# B&R Automation Studio project RobotComau
Automation Studio 4.11.3.51 SP; technology packages: mapp 5.18.0, mappCockpit 5.18.0, mappMotion 5.18.1, mappView 5.18.1, mappVision 5.18.0

## Configuration Config1

CPU 5APC3100.KBU1-000, AutomationRuntime B4.92, Build 4.1.2, Safety 0.0, Vc V4.72.5

### Task classes (Cpu.sw)
```
Cyclic#1 (cycle 2000 us, tolerance 0 us):
  OpcCtrl <- Services.OpcCtrl.prg
  ComauManua <- Robot.PackML.PackML_Manual.prg
  PackML_Aut <- Robot.PackML.PackML_Auto.prg
  PackML_Log <- Robot.PackML.PackML_Logic.prg
  PackML_Sem <- Robot.PackML.PackML_SemiAuto.prg
  RobotMove <- (binary)
Cyclic#2:
  File_explo <- Services.File_explorer.prg
Cyclic#4:
  Alarms <- Services.Alarms.prg
  Elements_d <- Camera.Elements_detection.prg
  Recipe <- Robot.Recipe.prg
  AuditProgr <- Services.AuditPckg.AuditProgram.prg
  AlarmClear <- Services.AlarmClearHistory.prg
DataObjects: McAcpSys
NcDataObjects: McDriveLog
Binaries: McAcpDrv, udbdef, McAcpSim, mvLoader, arflatprv, McPathXT, TCData, visionUnit, mCoWebSc, McMechSys, FWRules, arcoal, arsvcreg, TCLang, Settings, iomap, Config_3, Settings_1, viComp, Config_4, Role, ashwac, Hierarchy, asfw, Config_5, sysconf, Config_2, arconfig, Config_1, ashwd, User, Config_6, Config, Config_7, Config_9, PixelCount, Config_8, Config_13, Config_11, Config_14, Config_12, Config_10, TC, viApp, Matching15
Libraries: McBase, ViBase, AsZip, FileIO, AsARCfg, powerlnk, AsEPL, AsIO, sys_lib, astime, runtime, MpRobotics, McAxGroup, MpBase, McPathGen, McAxis, McProgInt, McAcpAx, CoTrace, standard, MpAlarmX, MpUserX, AsArSdm, MpRecipe, MpAudit, asarprof, asieccon, asarlog, asmem, brsystem, dataobj, arssl, asopcuac, aseth, ashw, arcert, aruser, asbrstr, mpfile, asusb, MpPackML, MpServer, MpWebXs
```

### Hardware
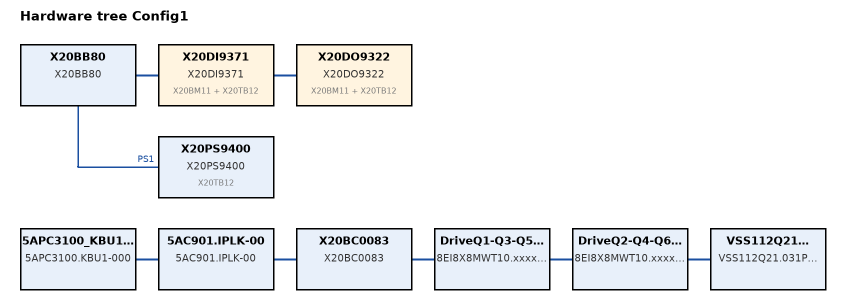
```
5AC901.IPLK-00 : 5AC901.IPLK-00 v1.8.0.1  [SL -> 5APC3100_KBU1_000.SL2]
  Connector IF1:
    MtuSize = 1500
    CycleTime = 400
    Channel1
    ChannelID1 = McAcpBroadcast
    ChannelType1 = OCTET[200]
    InternetAddress = 192.168.200.240
    SubnetMask = 255.255.255.0
5APC3100_KBU1_000 : 5APC3100.KBU1-000 v2.2.1.0
  Connector IF3:
    AssignedOperatingSystem = ARemb
    ActivateDevice = 1
    Mode = Manual
    InternetAddress = 192.168.0.10
    SubnetMask = 255.255.255.0
    InaPort = 81
    ActivateSnmp = 2
  Connector IF4:
    AssignedOperatingSystem = ARemb
    ActivateDevice = 1
  Connector IF5:
    AssignedOperatingSystem = ARemb
  Connector IF6:
    AssignedOperatingSystem = ARemb
  Connector IF7:
    AssignedOperatingSystem = ARemb
  Connector IF8:
    AssignedOperatingSystem = ARemb
  ConfigurationID = RobotComau_Config1
  RemMemDevice = PCI.2.IPLK.SRAM
  RemMemSize = 1024
  PermanentPvSize = 512
  RemanentGlobalPvSize = 512
  TimerDeviceType = EPLX2X
  TimerDevice = 5AC901.IPLK-00.IF1
  TaskClassIdleTime = 2000
  Cyclic1Duration = 2000
  Cyclic1Tolerance = 0
  FileDevice1
  FileDeviceName1 = CNC_PrgDir
  FileDevicePath1 = F:\RobotProgram
  FileDevice2
  FileDeviceName2 = RecipeDir
  FileDevicePath2 = F:\Data
  FileDevice3
  FileDeviceName3 = AuditDir
  FileDevicePath3 = F:\Audit
  FileDevice4
  FileDeviceName4 = FilesDir
  FileDevicePath4 = F:\
  FtpUser1
  FtpUsername1 = admin
  FtpUserPassword1 = QCzPEyxrRcQJkbJUmFYJydudCaTwVAMxyUFRcNQN44M=
  FtpUserSalt1 = 07CFXo9y
  FTPAccessRight1 = 0
  ActivateOpcUa = 1
  OpcUaActivateAuditEvents = 1
  OpcUa_Security_AdminRole = Administrators
  OpcUaInformationModels_PV_Version = 1
DriveQ1-Q3-Q5_Racer3_1 : 8EI8X8MWT10.xxxx-1 v2.3.1.1  [PLK1 -> X20BC0083.PLK2 (NodeNumber=4) [Cable Type=PowerlinkCable, Length=10, Version=1.0.0.3]; PLK2 -> DriveQ2-Q4-Q6_Racer3_1.PLK1 (NodeNumber=4) [Cable Type=PowerlinkCable, Length=10, Version=1.0.0.3]]
  DriveConfiguration/Module:
    McAcoposTypeID = AcoposP3TConfig
    ActivateACOPOSSimulationOnPLC = 0
  DriveConfiguration/Encoder/EncoderX41:
    InterfaceType = EnDat
  DriveConfiguration/Encoder/EncoderX42:
    InterfaceType = EnDat
  DriveConfiguration/Encoder/EncoderX43:
    InterfaceType = EnDat
  DriveConfiguration/Channel[1]/RealAxis:
    AxisReference = gAxisQ1_Racer3_1
    MechanicalElementsIsInvisible = 0
  DriveConfiguration/Channel[1]/RealAxis/MechanicalElements/Gearbox:
    InputIsReadOnly = 1
    Input = 81818
    OutputIsReadOnly = 1
    Output = 1000
  DriveConfiguration/Channel[1]/RealAxis/MechanicalElements/RotaryToLinearTransformation:
    ReferenceDistanceIsReadOnly = 1
    ReferenceDistance = 360
  DriveConfiguration/Channel[1]/RealAxis/Controller:
    ModeIsReadOnly = 1
    Mode = PositionControllerWithTorqueFeedForward
  DriveConfiguration/Channel[1]/RealAxis/Controller/Mode/Position:
    ProportionalGainIsReadOnly = 1
    ProportionalGain = 75.0
    IntegrationTimeIsReadOnly = 1
    IntegrationTime = 0.0
    TotalDelayTime = 0.0004
  DriveConfiguration/Channel[1]/RealAxis/Controller/Mode/Speed:
    ProportionalGainIsReadOnly = 1
    ProportionalGain = 2.0
    IntegrationTimeIsReadOnly = 1
    IntegrationTime = 0.0
    FilterTimeIsReadOnly = 1
    FilterTime = 0.0008
  DriveConfiguration/Channel[1]/RealAxis/Controller/Mode:
    FeedForwardIsReadOnly = 1
    FeedForward = CyclicValueFromAxesGroup
  DriveConfiguration/Channel[1]/RealAxis/Controller/Mode/LoopFilters:
    LoopFilterXIsReadOnly = 0
    LoopFilter1 = NotUsed
    LoopFilter2 = NotUsed
    LoopFilter3 = NotUsed
  DriveConfiguration/Channel[1]/RealAxis/Homing:
    ModeIsReadOnly = 0
    Mode = RestorePosition
    RestorePositionVariable = ::RestorePos[0]
  DriveConfiguration/Channel[1]/RealAxis/StopReaction:
    QuickstopIsReadOnly = 0
    Quickstop = DecelerationLimit
    DriveErrorIsReadOnly = 0
    DriveError = DecelerationLimit
  DriveConfiguration/Channel[1]/RealAxis/MovementErrorLimits:
    PositionError = 1.0
    VelocityErrorMonitoring = Automatic1
  DriveConfiguration/Channel[1]/RealAxis:
    JerkFilterIsReadOnly = 0
    JerkFilter = Used
  DriveConfiguration/Channel[1]/RealAxis/JerkFilter:
    JerkTimeMin = 0
    JerkTime = 0.01
  DriveConfiguration/Channel[1]/RealAxis/DigitalInputs/HomingSwitch:
    SourceIsReadOnly = 0
    Source = NotUsed
    Level = High
  DriveConfiguration/Channel[1]/RealAxis/DigitalInputs/PositiveLimitSwitch:
    SourceIsReadOnly = 0
    Source = NotUsed
    Level = High
  DriveConfiguration/Channel[1]/RealAxis/DigitalInputs/NegativeLimitSwitch:
    SourceIsReadOnly = 0
    Source = NotUsed
    Level = High
  DriveConfiguration/Channel[1]/RealAxis/DigitalInputs/Trigger1:
    Source = X8Trigger1
    Level = High
  DriveConfiguration/Channel[1]/RealAxis/DigitalInputs/Trigger2:
    Source = X8Trigger2
    Level = High
  DriveConfiguration/Channel[1]/RealAxis/DigitalInputs/Quickstop:
    Input = Trigger2
  DriveConfiguration/Channel[1]/RealAxis/Simulation:
    SimulationModeOnPLC = SetValueGeneration
    SimulationModeOnACOPOS = NotUsed
  DriveConfiguration/Channel[1]/RealAxis/AxisFeatures:
    FeatureRef[1] = Feature_Brake_Racer3_1
  DriveConfiguration/Channel[1]:
    ExternalEncoderAxis = NotUsed
  DriveConfiguration/Channel[2]/RealAxis:
    AxisReference = gAxisQ3_Racer3_1
    MechanicalElementsIsInvisible = 0
  DriveConfiguration/Channel[2]/RealAxis/MechanicalElements/Gearbox:
    InputIsReadOnly = 1
    Input = 72
    OutputIsReadOnly = 1
    Output = 1
  DriveConfiguration/Channel[2]/RealAxis/MechanicalElements/RotaryToLinearTransformation:
    ReferenceDistanceIsReadOnly = 1
    ReferenceDistance = 360
  DriveConfiguration/Channel[2]/RealAxis/Controller:
    ModeIsReadOnly = 1
    Mode = PositionControllerWithTorqueFeedForward
  DriveConfiguration/Channel[2]/RealAxis/Controller/Mode/Position:
    ProportionalGainIsReadOnly = 1
    ProportionalGain = 50.0
    IntegrationTimeIsReadOnly = 1
    IntegrationTime = 0.0
    TotalDelayTime = 0.0004
  DriveConfiguration/Channel[2]/RealAxis/Controller/Mode/Speed:
    ProportionalGainIsReadOnly = 1
    ProportionalGain = 1.5
    IntegrationTimeIsReadOnly = 1
    IntegrationTime = 0.0
    FilterTimeIsReadOnly = 1
    FilterTime = 0.0008
  DriveConfiguration/Channel[2]/RealAxis/Controller/Mode:
    FeedForwardIsReadOnly = 1
    FeedForward = CyclicValueFromAxesGroup
  DriveConfiguration/Channel[2]/RealAxis/Controller/Mode/LoopFilters:
    LoopFilterXIsReadOnly = 0
    LoopFilter1 = NotUsed
    LoopFilter2 = NotUsed
    LoopFilter3 = NotUsed
  DriveConfiguration/Channel[2]/RealAxis/Homing:
    ModeIsReadOnly = 0
    Mode = RestorePosition
    RestorePositionVariable = ::RestorePos[2]
  DriveConfiguration/Channel[2]/RealAxis/StopReaction:
    QuickstopIsReadOnly = 0
    Quickstop = DecelerationLimit
    DriveErrorIsReadOnly = 0
    DriveError = DecelerationLimit
  DriveConfiguration/Channel[2]/RealAxis/MovementErrorLimits:
    PositionError = 1.0
    VelocityErrorMonitoring = Automatic1
  DriveConfiguration/Channel[2]/RealAxis:
    JerkFilterIsReadOnly = 0
    JerkFilter = Used
  DriveConfiguration/Channel[2]/RealAxis/JerkFilter:
    JerkTimeMin = 0
    JerkTime = 0.01
  DriveConfiguration/Channel[2]/RealAxis/DigitalInputs/HomingSwitch:
    SourceIsReadOnly = 0
    Source = NotUsed
    Level = High
  DriveConfiguration/Channel[2]/RealAxis/DigitalInputs/PositiveLimitSwitch:
    SourceIsReadOnly = 0
    Source = NotUsed
    Level = High
  DriveConfiguration/Channel[2]/RealAxis/DigitalInputs/NegativeLimitSwitch:
    SourceIsReadOnly = 0
    Source = NotUsed
    Level = High
  DriveConfiguration/Channel[2]/RealAxis/DigitalInputs/Trigger1:
    Source = X8Trigger1
    Level = High
  DriveConfiguration/Channel[2]/RealAxis/DigitalInputs/Trigger2:
    Source = X8Trigger2
    Level = High
  DriveConfiguration/Channel[2]/RealAxis/DigitalInputs/Quickstop:
    Input = Trigger2
  DriveConfiguration/Channel[2]/RealAxis/Simulation:
    SimulationModeOnPLC = SetValueGeneration
    SimulationModeOnACOPOS = NotUsed
  DriveConfiguration/Channel[2]/RealAxis/AxisFeatures:
    FeatureRef[1] = Feature_Brake_Racer3_1
  DriveConfiguration/Channel[2]:
    ExternalEncoderAxis = NotUsed
  DriveConfiguration/Channel[3]/RealAxis:
    AxisReference = gAxisQ5_Racer3_1
    MechanicalElementsIsInvisible = 0
  DriveConfiguration/Channel[3]/RealAxis/MechanicalElements/Gearbox:
    InputIsReadOnly = 1
    Input = 612
    OutputIsReadOnly = 1
    Output = 10
  DriveConfiguration/Channel[3]/RealAxis/MechanicalElements/RotaryToLinearTransformation:
    ReferenceDistanceIsReadOnly = 1
    ReferenceDistance = 360
  DriveConfiguration/Channel[3]/RealAxis/Controller:
    ModeIsReadOnly = 1
    Mode = PositionControllerWithTorqueFeedForward
  DriveConfiguration/Channel[3]/RealAxis/Controller/Mode/Position:
    ProportionalGainIsReadOnly = 1
    ProportionalGain = 200.0
    IntegrationTimeIsReadOnly = 1
    IntegrationTime = 0.0
    TotalDelayTime = 0.0004
  DriveConfiguration/Channel[3]/RealAxis/Controller/Mode/Speed:
    ProportionalGainIsReadOnly = 1
    ProportionalGain = 1.5
    IntegrationTimeIsReadOnly = 1
    IntegrationTime = 0.0
    FilterTimeIsReadOnly = 1
    FilterTime = 0.0008
  DriveConfiguration/Channel[3]/RealAxis/Controller/Mode:
    FeedForwardIsReadOnly = 1
    FeedForward = CyclicValueFromAxesGroup
  DriveConfiguration/Channel[3]/RealAxis/Controller/Mode/LoopFilters:
    LoopFilterXIsReadOnly = 0
    LoopFilter1 = NotUsed
    LoopFilter2 = NotUsed
    LoopFilter3 = NotUsed
  DriveConfiguration/Channel[3]/RealAxis/Homing:
    ModeIsReadOnly = 0
    Mode = RestorePosition
    RestorePositionVariable = ::RestorePos[4]
  DriveConfiguration/Channel[3]/RealAxis/StopReaction:
    QuickstopIsReadOnly = 0
    Quickstop = DecelerationLimit
    DriveErrorIsReadOnly = 0
    DriveError = DecelerationLimit
  DriveConfiguration/Channel[3]/RealAxis/MovementErrorLimits:
    PositionError = 1.0
    VelocityErrorMonitoring = Automatic1
  DriveConfiguration/Channel[3]/RealAxis:
    JerkFilterIsReadOnly = 0
    JerkFilter = Used
  DriveConfiguration/Channel[3]/RealAxis/JerkFilter:
    JerkTimeMin = 0
    JerkTime = 0.01
  DriveConfiguration/Channel[3]/RealAxis/DigitalInputs/HomingSwitch:
    SourceIsReadOnly = 0
    Source = NotUsed
    Level = High
  DriveConfiguration/Channel[3]/RealAxis/DigitalInputs/PositiveLimitSwitch:
    SourceIsReadOnly = 0
    Source = NotUsed
    Level = High
  DriveConfiguration/Channel[3]/RealAxis/DigitalInputs/NegativeLimitSwitch:
    SourceIsReadOnly = 0
    Source = NotUsed
    Level = High
  DriveConfiguration/Channel[3]/RealAxis/DigitalInputs/Trigger1:
    Source = X8Trigger1
    Level = High
  DriveConfiguration/Channel[3]/RealAxis/DigitalInputs/Trigger2:
    Source = X8Trigger2
    Level = High
  DriveConfiguration/Channel[3]/RealAxis/DigitalInputs/Quickstop:
    Input = Trigger2
  DriveConfiguration/Channel[3]/RealAxis/Simulation:
    SimulationModeOnPLC = SetValueGeneration
    SimulationModeOnACOPOS = NotUsed
  DriveConfiguration/Channel[3]/RealAxis/AxisFeatures:
    FeatureRef[1] = Feature_Brake_Racer3_1
  DriveConfiguration/Channel[3]:
    ExternalEncoderAxis = NotUsed
DriveQ2-Q4-Q6_Racer3_1 : 8EI8X8MWT10.xxxx-1 v2.3.1.1  [PLK1 -> DriveQ1-Q3-Q5_Racer3_1.PLK2 (NodeNumber=5) [Cable Type=PowerlinkCable, Length=10, Version=1.0.0.3]; PLK2 -> VSS112Q21.031P-000.PLK2 (NodeNumber=5) [Cable Type=PowerlinkCable, Length=10, Version=1.0.0.3]]
  DriveConfiguration/Module:
    McAcoposTypeID = AcoposP3TConfig
    ActivateACOPOSSimulationOnPLC = 0
  DriveConfiguration/Encoder/EncoderX41:
    InterfaceType = EnDat
  DriveConfiguration/Encoder/EncoderX42:
    InterfaceType = EnDat
  DriveConfiguration/Encoder/EncoderX43:
    InterfaceType = EnDat
  DriveConfiguration/Channel[1]/RealAxis:
    AxisReference = gAxisQ2_Racer3_1
    MechanicalElementsIsInvisible = 0
  DriveConfiguration/Channel[1]/RealAxis/MechanicalElements/Gearbox:
    InputIsReadOnly = 1
    Input = 80
    OutputIsReadOnly = 1
    Output = 1
  DriveConfiguration/Channel[1]/RealAxis/MechanicalElements/RotaryToLinearTransformation:
    ReferenceDistanceIsReadOnly = 1
    ReferenceDistance = 360
  DriveConfiguration/Channel[1]/RealAxis/Controller:
    ModeIsReadOnly = 1
    Mode = PositionControllerWithTorqueFeedForward
  DriveConfiguration/Channel[1]/RealAxis/Controller/Mode/Position:
    ProportionalGainIsReadOnly = 1
    ProportionalGain = 50.0
    IntegrationTimeIsReadOnly = 1
    IntegrationTime = 0.0
    TotalDelayTime = 0.0004
  DriveConfiguration/Channel[1]/RealAxis/Controller/Mode/Speed:
    ProportionalGainIsReadOnly = 1
    ProportionalGain = 2.0
    IntegrationTimeIsReadOnly = 1
    IntegrationTime = 0.0
    FilterTimeIsReadOnly = 1
    FilterTime = 0.0008
  DriveConfiguration/Channel[1]/RealAxis/Controller/Mode:
    FeedForwardIsReadOnly = 1
    FeedForward = CyclicValueFromAxesGroup
  DriveConfiguration/Channel[1]/RealAxis/Controller/Mode/LoopFilters:
    LoopFilterXIsReadOnly = 0
    LoopFilter1 = NotUsed
    LoopFilter2 = NotUsed
    LoopFilter3 = NotUsed
  DriveConfiguration/Channel[1]/RealAxis/Homing:
    ModeIsReadOnly = 0
    Mode = RestorePosition
    RestorePositionVariable = ::RestorePos[1]
  DriveConfiguration/Channel[1]/RealAxis/StopReaction:
    QuickstopIsReadOnly = 0
    Quickstop = DecelerationLimit
    DriveErrorIsReadOnly = 0
    DriveError = DecelerationLimit
  DriveConfiguration/Channel[1]/RealAxis/MovementErrorLimits:
    PositionError = 1.0
    VelocityErrorMonitoring = Automatic1
  DriveConfiguration/Channel[1]/RealAxis:
    JerkFilterIsReadOnly = 0
    JerkFilter = Used
  DriveConfiguration/Channel[1]/RealAxis/JerkFilter:
    JerkTimeMin = 0
    JerkTime = 0.01
  DriveConfiguration/Channel[1]/RealAxis/DigitalInputs/HomingSwitch:
    SourceIsReadOnly = 0
    Source = NotUsed
    Level = High
  DriveConfiguration/Channel[1]/RealAxis/DigitalInputs/PositiveLimitSwitch:
    SourceIsReadOnly = 0
    Source = NotUsed
    Level = High
  DriveConfiguration/Channel[1]/RealAxis/DigitalInputs/NegativeLimitSwitch:
    SourceIsReadOnly = 0
    Source = NotUsed
    Level = High
  DriveConfiguration/Channel[1]/RealAxis/DigitalInputs/Trigger1:
    Source = X8Trigger1
    Level = High
  DriveConfiguration/Channel[1]/RealAxis/DigitalInputs/Trigger2:
    Source = X8Trigger2
    Level = High
  DriveConfiguration/Channel[1]/RealAxis/DigitalInputs/Quickstop:
    Input = Trigger2
  DriveConfiguration/Channel[1]/RealAxis/Simulation:
    SimulationModeOnPLC = SetValueGeneration
    SimulationModeOnACOPOS = NotUsed
  DriveConfiguration/Channel[1]/RealAxis/AxisFeatures:
    FeatureRef[1] = Feature_Brake_Racer3_1
  DriveConfiguration/Channel[1]:
    ExternalEncoderAxis = NotUsed
  DriveConfiguration/Channel[2]/RealAxis:
    AxisReference = gAxisQ4_Racer3_1
    MechanicalElementsIsInvisible = 0
  DriveConfiguration/Channel[2]/RealAxis/MechanicalElements/Gearbox:
    InputIsReadOnly = 1
    Input = 612
    OutputIsReadOnly = 1
    Output = 10
  DriveConfiguration/Channel[2]/RealAxis/MechanicalElements/RotaryToLinearTransformation:
    ReferenceDistanceIsReadOnly = 1
    ReferenceDistance = 360
  DriveConfiguration/Channel[2]/RealAxis/Controller:
    ModeIsReadOnly = 1
    Mode = PositionControllerWithTorqueFeedForward
  DriveConfiguration/Channel[2]/RealAxis/Controller/Mode/Position:
    ProportionalGainIsReadOnly = 1
    ProportionalGain = 100.0
    IntegrationTimeIsReadOnly = 1
    IntegrationTime = 0.0
    TotalDelayTime = 0.0004
  DriveConfiguration/Channel[2]/RealAxis/Controller/Mode/Speed:
    ProportionalGainIsReadOnly = 1
    ProportionalGain = 2.0
    IntegrationTimeIsReadOnly = 1
    IntegrationTime = 0.0
    FilterTimeIsReadOnly = 1
    FilterTime = 0.0008
  DriveConfiguration/Channel[2]/RealAxis/Controller/Mode:
    FeedForwardIsReadOnly = 1
    FeedForward = CyclicValueFromAxesGroup
  DriveConfiguration/Channel[2]/RealAxis/Controller/Mode/LoopFilters:
    LoopFilterXIsReadOnly = 0
    LoopFilter1 = NotUsed
    LoopFilter2 = NotUsed
    LoopFilter3 = NotUsed
  DriveConfiguration/Channel[2]/RealAxis/Homing:
    ModeIsReadOnly = 0
    Mode = RestorePosition
    RestorePositionVariable = ::RestorePos[3]
  DriveConfiguration/Channel[2]/RealAxis/StopReaction:
    QuickstopIsReadOnly = 0
    Quickstop = DecelerationLimit
    DriveErrorIsReadOnly = 0
    DriveError = DecelerationLimit
  DriveConfiguration/Channel[2]/RealAxis/MovementErrorLimits:
    PositionError = 1.0
    VelocityErrorMonitoring = Automatic1
  DriveConfiguration/Channel[2]/RealAxis:
    JerkFilterIsReadOnly = 0
    JerkFilter = Used
  DriveConfiguration/Channel[2]/RealAxis/JerkFilter:
    JerkTimeMin = 0
    JerkTime = 0.01
  DriveConfiguration/Channel[2]/RealAxis/DigitalInputs/HomingSwitch:
    SourceIsReadOnly = 0
    Source = NotUsed
    Level = High
  DriveConfiguration/Channel[2]/RealAxis/DigitalInputs/PositiveLimitSwitch:
    SourceIsReadOnly = 0
    Source = NotUsed
    Level = High
  DriveConfiguration/Channel[2]/RealAxis/DigitalInputs/NegativeLimitSwitch:
    SourceIsReadOnly = 0
    Source = NotUsed
    Level = High
  DriveConfiguration/Channel[2]/RealAxis/DigitalInputs/Trigger1:
    Source = X8Trigger1
    Level = High
  DriveConfiguration/Channel[2]/RealAxis/DigitalInputs/Trigger2:
    Source = X8Trigger2
    Level = High
  DriveConfiguration/Channel[2]/RealAxis/DigitalInputs/Quickstop:
    Input = Trigger2
  DriveConfiguration/Channel[2]/RealAxis/Simulation:
    SimulationModeOnPLC = SetValueGeneration
    SimulationModeOnACOPOS = NotUsed
  DriveConfiguration/Channel[2]/RealAxis/AxisFeatures:
    FeatureRef[1] = Feature_Brake_Racer3_1
  DriveConfiguration/Channel[2]:
    ExternalEncoderAxis = NotUsed
  DriveConfiguration/Channel[3]/RealAxis:
    AxisReference = gAxisQ6_Racer3_1
    MechanicalElementsIsInvisible = 0
  DriveConfiguration/Channel[3]/RealAxis/MechanicalElements/Gearbox:
    InputIsReadOnly = 1
    Input = 40
    OutputIsReadOnly = 1
    Output = 1
  DriveConfiguration/Channel[3]/RealAxis/MechanicalElements/RotaryToLinearTransformation:
    ReferenceDistanceIsReadOnly = 1
    ReferenceDistance = 360
  DriveConfiguration/Channel[3]/RealAxis/Controller:
    ModeIsReadOnly = 1
    Mode = PositionControllerWithTorqueFeedForward
  DriveConfiguration/Channel[3]/RealAxis/Controller/Mode/Position:
    ProportionalGainIsReadOnly = 1
    ProportionalGain = 200.0
    IntegrationTimeIsReadOnly = 1
    IntegrationTime = 0.0
    TotalDelayTime = 0.0004
  DriveConfiguration/Channel[3]/RealAxis/Controller/Mode/Speed:
    ProportionalGainIsReadOnly = 1
    ProportionalGain = 1.5
    IntegrationTimeIsReadOnly = 1
    IntegrationTime = 0.0
    FilterTimeIsReadOnly = 1
    FilterTime = 0.0008
  DriveConfiguration/Channel[3]/RealAxis/Controller/Mode:
    FeedForwardIsReadOnly = 1
    FeedForward = CyclicValueFromAxesGroup
  DriveConfiguration/Channel[3]/RealAxis/Controller/Mode/LoopFilters:
    LoopFilterXIsReadOnly = 0
    LoopFilter1 = NotUsed
    LoopFilter2 = NotUsed
    LoopFilter3 = NotUsed
  DriveConfiguration/Channel[3]/RealAxis/Homing:
    ModeIsReadOnly = 0
    Mode = RestorePosition
    RestorePositionVariable = ::RestorePos[5]
  DriveConfiguration/Channel[3]/RealAxis/StopReaction:
    QuickstopIsReadOnly = 0
    Quickstop = DecelerationLimit
    DriveErrorIsReadOnly = 0
    DriveError = DecelerationLimit
  DriveConfiguration/Channel[3]/RealAxis/MovementErrorLimits:
    PositionError = 1.0
    VelocityErrorMonitoring = Automatic1
  DriveConfiguration/Channel[3]/RealAxis:
    JerkFilterIsReadOnly = 0
    JerkFilter = Used
  DriveConfiguration/Channel[3]/RealAxis/JerkFilter:
    JerkTimeMin = 0
    JerkTime = 0.01
  DriveConfiguration/Channel[3]/RealAxis/DigitalInputs/HomingSwitch:
    SourceIsReadOnly = 0
    Source = NotUsed
    Level = High
  DriveConfiguration/Channel[3]/RealAxis/DigitalInputs/PositiveLimitSwitch:
    SourceIsReadOnly = 0
    Source = NotUsed
    Level = High
  DriveConfiguration/Channel[3]/RealAxis/DigitalInputs/NegativeLimitSwitch:
    SourceIsReadOnly = 0
    Source = NotUsed
    Level = High
  DriveConfiguration/Channel[3]/RealAxis/DigitalInputs/Trigger1:
    Source = X8Trigger1
    Level = High
  DriveConfiguration/Channel[3]/RealAxis/DigitalInputs/Trigger2:
    Source = X8Trigger2
    Level = High
  DriveConfiguration/Channel[3]/RealAxis/DigitalInputs/Quickstop:
    Input = Trigger2
  DriveConfiguration/Channel[3]/RealAxis/Simulation:
    SimulationModeOnPLC = SetValueGeneration
    SimulationModeOnACOPOS = NotUsed
  DriveConfiguration/Channel[3]/RealAxis/AxisFeatures:
    FeatureRef[1] = Feature_Brake_Racer3_1
  DriveConfiguration/Channel[3]:
    ExternalEncoderAxis = NotUsed
VSS112Q21.031P-000 : VSS112Q21.031P-000 v1.6.0.543  [PLK2 -> DriveQ2-Q4-Q6_Racer3_1.PLK2 (NodeNumber=6) [Cable Type=PowerlinkCable, Length=10, Version=1.0.0.3]]
  VisionConfig = gCamera
X20BB80 : X20BB80 v1.1.0.0
X20BC0083 : X20BC0083 v2.12.0.0  [PLK1 -> 5AC901.IPLK-00.IF1 (NodeNumber=3) [Cable Type=PowerlinkCable, Length=10, Version=1.0.0.3]; PLK2 -> DriveQ1-Q3-Q5_Racer3_1.PLK1 (NodeNumber=3) [Cable Type=PowerlinkCable, Length=10, Version=1.0.0.3]; SL -> X20BB80.SL1]
X20BM11 : X20BM11 v1.1.0.0  [X2X1 -> X20BB80.IF1]
X20BM11a : X20BM11 v1.1.0.0  [X2X1 -> X20BM11.X2X2]
X20DI9371 : X20DI9371 v1.3.0.0  [SS1 -> X20TB12a.SS; SL -> X20BM11.SL1]
X20DO9322 : X20DO9322 v1.4.0.0  [SS1 -> X20TB12b.SS; SL -> X20BM11a.SL1]
X20PS9400 : X20PS9400 v1.7.0.0  [SS1 -> X20TB12.SS; PS -> X20BB80.PS1]
X20TB12 : X20TB12 v1.0.0.0
X20TB12a : X20TB12 v1.0.0.0
X20TB12b : X20TB12 v1.0.0.0
```

### IoMap.iom - 5APC3100_KBU1_000/IoMap.iom
```iecst
VAR_CONFIG
	::Camera_0.ImageAcq AT %QX."VSS112Q21.031P-000".ImageAcquisition;
	::Camera_0.PixelCntSquareArray[0] AT %ID."VSS112Q21.031P-000".FoundedPixelsNum01;
	::Camera_0.PixelCntSquareArray[1] AT %ID."VSS112Q21.031P-000".FoundedPixelsNum02;
	::Camera_0.PixelCntSquareArray[2] AT %ID."VSS112Q21.031P-000".FoundedPixelsNum03;
	::Camera_0.PixelCntSquareArray[3] AT %ID."VSS112Q21.031P-000".FoundedPixelsNum04;
	::Camera_0.PixelCntSquareArray[4] AT %ID."VSS112Q21.031P-000".FoundedPixelsNum05;
	::Camera_0.PixelCntSquareArray[5] AT %ID."VSS112Q21.031P-000".FoundedPixelsNum06;
	::Camera_0.PixelCntSquareArray[6] AT %ID."VSS112Q21.031P-000".FoundedPixelsNum07;
	::Camera_0.PixelCntSquareArray[7] AT %ID."VSS112Q21.031P-000".FoundedPixelsNum08;
	::Camera_0.PixelCntSquareArray[8] AT %ID."VSS112Q21.031P-000".FoundedPixelsNum09;
	::Camera_0.PixelCntSquareArray[9] AT %ID."VSS112Q21.031P-000".FoundedPixelsNum10;
	::Camera_0.PixelCntSquareArray[10] AT %ID."VSS112Q21.031P-000".FoundedPixelsNum11;
	::Camera_0.PixelCntSquareArray[11] AT %ID."VSS112Q21.031P-000".FoundedPixelsNum12;
	::Camera_0.PixelCntSquareArray[12] AT %ID."VSS112Q21.031P-000".FoundedPixelsNum13;
	::Camera_0.PixelCntSquareArray[13] AT %ID."VSS112Q21.031P-000".FoundedPixelsNum14;
	::Camera_0.Focus AT %QW."VSS112Q21.031P-000".SetFocus;
	::Camera_0.ExposureTime AT %QD."VSS112Q21.031P-000".ExposureTime01;
	::Camera_0.Enable AT %QX."VSS112Q21.031P-000".EnableVF1;
	::Camera_0.NumSearch AT %QB."VSS112Q21.031P-000".NumSearch;
	::Camera_0.Ready AT %IX."VSS112Q21.031P-000".ImageAcquisitionReady;
	::Camera_0.FlashColor AT %QB."VSS112Q21.031P-000".FlashColor01;
	::Camera_0.FlashSegment AT %QB."VSS112Q21.031P-000".FlashSegment01;
	::Camera_0.ModelNumArray[0] AT %IB."VSS112Q21.031P-000".ModelNum01;
	::Camera_0.ModelNumArray[1] AT %IB."VSS112Q21.031P-000".ModelNum02;
	::Camera_0.ModelNumArray[2] AT %IB."VSS112Q21.031P-000".ModelNum03;
	::Camera_0.ModelNumArray[3] AT %IB."VSS112Q21.031P-000".ModelNum04;
	::Camera_0.ModelNumArray[4] AT %IB."VSS112Q21.031P-000".ModelNum05;
	::Camera_0.ModelNumArray[5] AT %IB."VSS112Q21.031P-000".ModelNum06;
	::Camera_0.ModelNumArray[6] AT %IB."VSS112Q21.031P-000".ModelNum07;
	::Camera_0.ModelNumArray[7] AT %IB."VSS112Q21.031P-000".ModelNum08;
	::Camera_0.ModelNumArray[8] AT %IB."VSS112Q21.031P-000".ModelNum09;
	::Camera_0.ModelNumArray[9] AT %IB."VSS112Q21.031P-000".ModelNum10;
	::Camera_0.ModelNumArray[10] AT %IB."VSS112Q21.031P-000".ModelNum11;
	::Camera_0.ModelNumArray[11] AT %IB."VSS112Q21.031P-000".ModelNum12;
	::Camera_0.ModelNumArray[12] AT %IB."VSS112Q21.031P-000".ModelNum13;
	::Camera_0.ModelNumArray[13] AT %IB."VSS112Q21.031P-000".ModelNum14;
	::doMagnet AT %QX."X20DO9322".DigitalOutput05;
	::Camera_0.ImgProcessingActive AT %IX."VSS112Q21.031P-000".ImageProcessingActive;
END_VAR
```

### Config_1.axesgroup - 5APC3100_KBU1_000/mappMotion/Comau_Racer3_1/Config_1.axesgroup
```
Element gAxesGroup_Racer3_1 (Type=axesgroup)
  Type = PathGenAxesGroup
    ProcessingTaskClass = 255
    License = 1
    PhysicalAxes:
      JointAxes:
        JointAxisAxisRefIsReadOnly = 0
        JointAxis[1]:
          Name = Q1
          AxisRef = gAxisQ1_Racer3_1
        JointAxis[2]:
          Name = Q2
          AxisRef = gAxisQ2_Racer3_1
        JointAxis[3]:
          Name = Q3
          AxisRef = gAxisQ3_Racer3_1
        JointAxis[4]:
          Name = Q4
          AxisRef = gAxisQ4_Racer3_1
        JointAxis[5]:
          Name = Q5
          AxisRef = gAxisQ5_Racer3_1
        JointAxis[6]:
          Name = Q6
          AxisRef = gAxisQ6_Racer3_1
    MechanicalSystem:
      MechSysRefIsReadOnly = 0
      MechSysRef = MechSys_Racer3_1
    BasicSettings:
      ModalDataBehaviour = ResetToDefault
      GeometryPlanning:
        TCPResolutionIsReadOnly = 0
        TCPResolution:
          LengthResolution = 0.001
          AngleResolution = 0.001
        RoundingMode = Standard
        MaxCornerDeviation = 0.0
        MaxTangentialTransitionDeviation = 0.05
        MaxRadiusDeviation = 0.001
        WorkingPlane = XY
      TrajectoryPlanningIsReadOnly = 0
      TrajectoryPlanning = Basic
        LimitCheckResolutionIsReadOnly = 0
        LimitCheckResolution = UserDefinedTime
          TimeIsReadOnly = 0
          Time = 0.005
        BufferTime = UserDefinedTime
          Time = 0.050
      Miscellaneous:
        NonMovementsLimit = NotUsed
    AxesGroupFeatures:
      FeatureRef[1] = Feature_Programs_Racer3_1
      FeatureRef[2] = Feature_FeedForward_Racer3_1
      FeatureRef[3] = Feature_Jogging_Racer3_1
      FeatureRef[4] = Feature_SharedBrakesSignals_Racer3_1
      FeatureRef[5] = Feature_WorkspaceMonitoring
  Alarms = MpAlarmX
```

### Config_2.axis - 5APC3100_KBU1_000/mappMotion/Comau_Racer3_1/Config_2.axis
```
Element gAxisQ1_Racer3_1 (Type=axis)
  BaseTypeIsReadOnly = 1
  BaseType = RotaryBounded
    MeasurementUnitIsReadOnly = 1
    MeasurementUnit = 17476
    MeasurementResolutionIsReadOnly = 1
    MeasurementResolution = 0.001
    CountDirectionIsReadOnly = 1
    CountDirection = Inverse
  MovementLimitsIsReadOnly = 1
  MovementLimits = InternalForPathControlledAxis
    Position:
      LowerLimitMin = -170.0
      UpperLimitMax = 170.0
      LowerLimit = -170.0
      UpperLimit = 170.0
    VelocityIsReadOnly = 1
    Velocity:
      VelocityMax = 420.0
      Velocity = 420.0
    AccelerationIsReadOnly = 1
    Acceleration:
      AccelerationMax = 1100.0
      Acceleration = 1100.0
    DecelerationIsReadOnly = 1
    Deceleration:
      DecelerationMax = 1100.0
      Deceleration = 1100.0
    JerkIsReadOnly = 1
    Jerk = Basic
      JerkMax = 3.4E38
      Jerk = 11000.0
    TorqueIsInvisible = 0
  Alarms = MpAlarmX
Element gAxisQ2_Racer3_1 (Type=axis)
  BaseTypeIsReadOnly = 1
  BaseType = RotaryBounded
    MeasurementUnitIsReadOnly = 1
    MeasurementUnit = 17476
    MeasurementResolutionIsReadOnly = 1
    MeasurementResolution = 0.001
    CountDirectionIsReadOnly = 1
    CountDirection = Standard
  MovementLimitsIsReadOnly = 1
  MovementLimits = InternalForPathControlledAxis
    Position:
      LowerLimitMin = -95.0
      UpperLimitMax = 135.0
      LowerLimit = -95.0
      UpperLimit = 135.0
    VelocityIsReadOnly = 1
    Velocity:
      VelocityMax = 450.0
      Velocity = 450.0
    AccelerationIsReadOnly = 1
    Acceleration:
      AccelerationMax = 750.0
      Acceleration = 750.0
    DecelerationIsReadOnly = 1
    Deceleration:
      DecelerationMax = 750.0
      Deceleration = 750.0
    JerkIsReadOnly = 1
    Jerk = Basic
      JerkMax = 3.4E38
      Jerk = 7500.0
    TorqueIsInvisible = 0
  Alarms = MpAlarmX
Element gAxisQ3_Racer3_1 (Type=axis)
  BaseTypeIsReadOnly = 1
  BaseType = RotaryBounded
    MeasurementUnitIsReadOnly = 1
    MeasurementUnit = 17476
    MeasurementResolutionIsReadOnly = 1
    MeasurementResolution = 0.001
    CountDirectionIsReadOnly = 1
    CountDirection = Inverse
  MovementLimitsIsReadOnly = 1
  MovementLimits = InternalForPathControlledAxis
    Position:
      LowerLimitMin = -155.0
      UpperLimitMax = 90.0
      LowerLimit = -155.0
      UpperLimit = 90.0
    VelocityIsReadOnly = 1
    Velocity:
      VelocityMax = 480.0
      Velocity = 480.0
    AccelerationIsReadOnly = 1
    Acceleration:
      AccelerationMax = 1250.0
      Acceleration = 1250.0
    DecelerationIsReadOnly = 1
    Deceleration:
      DecelerationMax = 1250.0
      Deceleration = 1250.0
    JerkIsReadOnly = 1
    Jerk = Basic
      JerkMax = 3.4E38
      Jerk = 12500.0
    TorqueIsInvisible = 0
  Alarms = MpAlarmX
Element gAxisQ4_Racer3_1 (Type=axis)
  BaseTypeIsReadOnly = 1
  BaseType = RotaryBounded
    MeasurementUnitIsReadOnly = 1
    MeasurementUnit = 17476
    MeasurementResolutionIsReadOnly = 1
    MeasurementResolution = 0.001
    CountDirectionIsReadOnly = 1
    CountDirection = Standard
  MovementLimitsIsReadOnly = 1
  MovementLimits = InternalForPathControlledAxis
    Position:
      LowerLimitMin = -200.0
      UpperLimitMax = 200.0
      LowerLimit = -200.0
      UpperLimit = 200.0
    VelocityIsReadOnly = 1
    Velocity:
      VelocityMax = 600.0
      Velocity = 600.0
    AccelerationIsReadOnly = 1
    Acceleration:
      AccelerationMax = 1200.0
      Acceleration = 1200.0
    DecelerationIsReadOnly = 1
    Deceleration:
      DecelerationMax = 1200.0
      Deceleration = 1200.0
    JerkIsReadOnly = 1
    Jerk = Basic
      JerkMax = 3.4E38
      Jerk = 12000.0
    TorqueIsInvisible = 0
  Alarms = MpAlarmX
Element gAxisQ5_Racer3_1 (Type=axis)
  BaseTypeIsReadOnly = 1
  BaseType = RotaryBounded
    MeasurementUnitIsReadOnly = 1
    MeasurementUnit = 17476
    MeasurementResolutionIsReadOnly = 1
    MeasurementResolution = 0.001
    CountDirectionIsReadOnly = 1
    CountDirection = Standard
  MovementLimitsIsReadOnly = 1
  MovementLimits = InternalForPathControlledAxis
    Position:
      LowerLimitMin = -125.0
      UpperLimitMax = 125.0
      LowerLimit = -125.0
      UpperLimit = 125.0
    VelocityIsReadOnly = 1
    Velocity:
      VelocityMax = 600.0
      Velocity = 600.0
    AccelerationIsReadOnly = 1
    Acceleration:
      AccelerationMax = 1200.0
      Acceleration = 1200.0
    DecelerationIsReadOnly = 1
    Deceleration:
      DecelerationMax = 1200.0
      Deceleration = 1200.0
    JerkIsReadOnly = 1
    Jerk = Basic
      JerkMax = 3.4E38
      Jerk = 12000.0
    TorqueIsInvisible = 0
  Alarms = MpAlarmX
Element gAxisQ6_Racer3_1 (Type=axis)
  BaseTypeIsReadOnly = 1
  BaseType = RotaryBounded
    MeasurementUnitIsReadOnly = 1
    MeasurementUnit = 17476
    MeasurementResolutionIsReadOnly = 1
    MeasurementResolution = 0.001
    CountDirectionIsReadOnly = 1
    CountDirection = Standard
  MovementLimitsIsReadOnly = 1
  MovementLimits = InternalForPathControlledAxis
    Position:
      LowerLimitMin = -2700.0
      UpperLimitMax = 2700.0
      LowerLimit = -2700.0
      UpperLimit = 2700.0
    VelocityIsReadOnly = 1
    Velocity:
      VelocityMax = 875.0
      Velocity = 875.0
    AccelerationIsReadOnly = 1
    Acceleration:
      AccelerationMax = 1800.0
      Acceleration = 1800.0
    DecelerationIsReadOnly = 1
    Deceleration:
      DecelerationMax = 1800.0
      Deceleration = 1800.0
    JerkIsReadOnly = 1
    Jerk = Basic
      JerkMax = 3.4E38
      Jerk = 18000.0
    TorqueIsInvisible = 0
  Alarms = MpAlarmX
```

### Config_3.mechanicalsystem - 5APC3100_KBU1_000/mappMotion/Comau_Racer3_1/Config_3.mechanicalsystem
```
Element MechSys_Racer3_1 (Type=mechanicalsystem)
  TypeIsReadOnly = 0
  Type = 6AxesRoboarm
    SubtypeIsReadOnly = 0
    Subtype = 6AxesRoboarmB
      DescriptionIsReadOnly = 0
      Description = Standard
        Dimensions:
          TranslationFromBaseToQ1IsReadOnly = 1
          TranslationFromBaseToQ1:
            X = 0.0
            Y = 0.0
            Z = 0.0
          TranslationFromQ1ToQ2IsReadOnly = 1
          TranslationFromQ1ToQ2:
            X = 50.0
            Y = 0.0
            Z = 365.0
          TranslationFromQ2ToQ3IsReadOnly = 1
          TranslationFromQ2ToQ3:
            X = 0.0
            Y = 0.0
            Z = 270.0
          TranslationFromQ3ToQ4IsReadOnly = 1
          TranslationFromQ3ToQ4:
            X = -50.0
            Y = 0.0
            Z = 0.0
          TranslationFromQ4ToQ5IsReadOnly = 1
          TranslationFromQ4ToQ5:
            Z = 305.94
          TranslationFromQ5ToQ6IsReadOnly = 1
          TranslationFromQ5ToQ6:
            Z = 0.0
          TranslationFromQ6ToFlangeIsReadOnly = 0
          TranslationFromQ6ToFlange:
            X = 0.0
            Y = 0.0
            Z = 80.0
        Offsets:
          JointAxisIsReadOnly = 1
          JointAxis[1] = 0.0
          JointAxis[2] = 0.0
          JointAxis[3] = 0.0
          JointAxis[4] = 0.0
          JointAxis[5] = 0.0
          JointAxis[6] = 0.0
        CountDirections:
          JointAxisIsReadOnly = 1
          JointAxis[1] = Inverse
          JointAxis[2] = Standard
          JointAxis[3] = Inverse
          JointAxis[4] = Inverse
          JointAxis[5] = Standard
          JointAxis[6] = Inverse
      CoordinatesNames = Default
        XCoordinateName = X
        YCoordinateName = Y
        ZCoordinateName = Z
        ACoordinateName = A
        BCoordinateName = B
        CCoordinateName = C
      WireFrameModelIsReadOnly = 0
      WireFrameModel = Standard
        Q1ToQ2IsReadOnly = 0
        Q1ToQ2 = ConnectionLine
          DistanceMin = -1.79769313486231E308
          DistanceMax = 1.79769313486231E308
          Distance = 0.0
        Q2ToQ3IsReadOnly = 0
        Q2ToQ3 = ConnectionLine
          DistanceMin = -1.79769313486231E308
          DistanceMax = 1.79769313486231E308
          Distance = 0.0
        Q3ToQ4IsReadOnly = 0
        Q3ToQ4 = ConnectionLine
          DistanceMin = -1.79769313486231E308
          DistanceMax = 1.79769313486231E308
          Distance = 0.0
        Q4ToQ5IsReadOnly = 0
        Q4ToQ5 = ConnectionLine
          DistanceMin = -1.79769313486231E308
          DistanceMax = 1.79769313486231E308
          Distance = 0.0
        Q5ToQ6IsReadOnly = 0
        Q5ToQ6 = ConnectionLine
          DistanceMin = -1.79769313486231E308
          DistanceMax = 1.79769313486231E308
          Distance = 0.0
        Q6ToFlangeIsReadOnly = 0
        Q6ToFlange = ConnectionLine
          DistanceMin = -1.79769313486231E308
          DistanceMax = 1.79769313486231E308
          Distance = 0.0
        FlangeToTcp = ConnectionLine
          DistanceMin = -1.79769313486231E308
          DistanceMax = 1.79769313486231E308
          Distance = 0.0
      DynamicModel = DynParTable
        TableRef
      InternalDynamicModelIsReadOnly = 0
      InternalDynamicModel = Used
        TypeIsReadOnly = 1
        Type = Comau Racer 3
        Row[1]:
          Index = 0
          Value = 4
          Unit = 
          Description = TRF_DYN11D_typ
        Row[2]:
          Index = 1
          Value = 0
          Unit = 
          Description = 
        Row[3]:
          Index = 2
          Value = 0
          Unit = 
          Description = 
        Row[4]:
          Index = 3
          Value = 0.99502
          Unit = kgm^2
          Description = m1*rc1x^2+m1*rc1y^2+Jzz1+(0.0025)*m2+m2*rc2y^2+(0.5)*Jxx2+(-0.5)*Jyy2+(0.5)*Jzz2+(0.0025)*m3+m3*rc3y^2+(0.5)*Jxx3+(-0.5)*Jyy3+(0.5)*Jzz3+(0.0025)*m4+(0.0025)*m5+(0.0025)*m6+(6694.1851)*JDrive1+(-3200)*JDrive2
        Row[5]:
          Index = 4
          Value = 0
          Unit = 
          Description = 
        Row[6]:
          Index = 5
          Value = 0
          Unit = 
          Description = 
        Row[7]:
          Index = 6
          Value = 0
          Unit = 
          Description = 
        Row[8]:
          Index = 7
          Value = -0.0079739
          Unit = kgm
          Description = m2*rc2x
        Row[9]:
          Index = 8
          Value = 0
          Unit = 
          Description = 
        Row[10]:
          Index = 9
          Value = 3.2569
          Unit = kgm
          Description = m2*rc2z+(0.27)*m3+(0.27)*m4+(0.27)*m5+(0.27)*m6
        Row[11]:
          Index = 10
          Value = -0.01529
          Unit = kgm^2
          Description = m2*rc2x*rc2y
        Row[12]:
          Index = 11
          Value = 0.018218
          Unit = kgm^2
          Description = m2*rc2y*rc2z+(0.27)*m3*rc3y
        Row[13]:
          Index = 12
          Value = -0.027
          Unit = kgm^2
          Description = m2*rc2x*rc2z
        Row[14]:
          Index = 13
          Value = 0.23153
          Unit = kgm^2
          Description = m2*rc2x^2+(-0.5)*Jxx2+(0.5)*Jyy2+(0.5)*Jzz2+(3200)*JDrive2
        Row[15]:
          Index = 14
          Value = 0
          Unit = 
          Description = 
        Row[16]:
          Index = 15
          Value = 1.1014
          Unit = kgm^2
          Description = m2*rc2z^2+(0.5)*Jxx2+(0.5)*Jyy2+(-0.5)*Jzz2+(0.0729)*m3+(0.0729)*m4+(0.0729)*m5+(0.0729)*m6+(3200)*JDrive2
        Row[17]:
          Index = 16
          Value = 0
          Unit = 
          Description = 
        Row[18]:
          Index = 17
          Value = 0
          Unit = 
          Description = 
        Row[19]:
          Index = 18
          Value = 0
          Unit = 
          Description = 
        Row[20]:
          Index = 19
          Value = 0
          Unit = 
          Description = 
        Row[21]:
          Index = 20
          Value = -0.32261
          Unit = kgm
          Description = m3*rc3x+(-0.05)*m4+(-0.05)*m5+(-0.05)*m6
        Row[22]:
          Index = 21
          Value = 0
          Unit = 
          Description = 
        Row[23]:
          Index = 22
          Value = 1.1289
          Unit = kgm
          Description = m3*rc3z+m4*rc4z+(0.30594)*m5+(0.30594)*m6
        Row[24]:
          Index = 23
          Value = -0.0059741
          Unit = kgm^2
          Description = m3*rc3x*rc3y
        Row[25]:
          Index = 24
          Value = 0.048102
          Unit = kgm^2
          Description = m3*rc3y*rc3z
        Row[26]:
          Index = 25
          Value = -0.049555
          Unit = kgm^2
          Description = m3*rc3x*rc3z+(-0.05)*m4*rc4z+(-0.015297)*m5+(-0.015297)*m6
        Row[27]:
          Index = 26
          Value = -0.026241
          Unit = kgm^2
          Description = m3*rc3x^2+(-0.5)*Jxx3+(0.5)*Jyy3+(0.5)*Jzz3+(0.0025)*m4+(0.0025)*m5+(0.0025)*m6
        Row[28]:
          Index = 27
          Value = 0
          Unit = 
          Description = 
        Row[29]:
          Index = 28
          Value = 0.21145
          Unit = kgm^2
          Description = m3*rc3z^2+(0.5)*Jxx3+(0.5)*Jyy3+(-0.5)*Jzz3+m4*rc4z^2+(0.5)*Jxx4+(0.5)*Jyy4+(-0.5)*Jzz4+(0.093599)*m5+(0.093599)*m6
        Row[30]:
          Index = 29
          Value = 0
          Unit = 
          Description = 
        Row[31]:
          Index = 30
          Value = 0
          Unit = 
          Description = 
        Row[32]:
          Index = 31
          Value = 0
          Unit = 
          Description = 
        Row[33]:
          Index = 32
          Value = 0
          Unit = 
          Description = 
        Row[34]:
          Index = 33
          Value = -0.0056373
          Unit = kgm
          Description = m4*rc4x
        Row[35]:
          Index = 34
          Value = 0.011806
          Unit = kgm
          Description = m4*rc4y+m5*rc5y
        Row[36]:
          Index = 35
          Value = 0
          Unit = 
          Description = 
        Row[37]:
          Index = 36
          Value = -0.0071612
          Unit = kgm^2
          Description = m4*rc4x*rc4y
        Row[38]:
          Index = 37
          Value = -0.00018934
          Unit = kgm^2
          Description = m4*rc4y*rc4z+(0.30594)*m5*rc5y
        Row[39]:
          Index = 38
          Value = 0.002269
          Unit = kgm^2
          Description = m4*rc4x*rc4z
        Row[40]:
          Index = 39
          Value = -0.0073563
          Unit = kgm^2
          Description = m4*rc4x^2+(-0.5)*Jxx4+(0.5)*Jyy4+(0.5)*Jzz4
        Row[41]:
          Index = 40
          Value = -0.00050442
          Unit = kgm^2
          Description = m4*rc4y^2+(0.5)*Jxx4+(-0.5)*Jyy4+(0.5)*Jzz4+m5*rc5y^2+(0.5)*Jxx5+(-0.5)*Jyy5+(0.5)*Jzz5
        Row[42]:
          Index = 41
          Value = 0
          Unit = 
          Description = 
        Row[43]:
          Index = 42
          Value = 0
          Unit = 
          Description = 
        Row[44]:
          Index = 43
          Value = 0
          Unit = 
          Description = 
        Row[45]:
          Index = 44
          Value = 0
          Unit = 
          Description = 
        Row[46]:
          Index = 45
          Value = 0
          Unit = 
          Description = 
        Row[47]:
          Index = 46
          Value = -0.0030729
          Unit = kgm
          Description = m5*rc5x
        Row[48]:
          Index = 47
          Value = 0
          Unit = 
          Description = 
        Row[49]:
          Index = 48
          Value = 0.0086628
          Unit = kgm
          Description = m5*rc5z+m6*rc6z
        Row[50]:
          Index = 49
          Value = 5.0384e-05
          Unit = kgm^2
          Description = m5*rc5x*rc5y
        Row[51]:
          Index = 50
          Value = 0.004449
          Unit = kgm^2
          Description = m5*rc5y*rc5z
        Row[52]:
          Index = 51
          Value = 0.00094987
          Unit = kgm^2
          Description = m5*rc5x*rc5z
        Row[53]:
          Index = 52
          Value = -0.0039698
          Unit = kgm^2
          Description = m5*rc5x^2+(-0.5)*Jxx5+(0.5)*Jyy5+(0.5)*Jzz5
        Row[54]:
          Index = 53
          Value = 0
          Unit = 
          Description = 
        Row[55]:
          Index = 54
          Value = -0.0023413
          Unit = kgm^2
          Description = m5*rc5z^2+(0.5)*Jxx5+(0.5)*Jyy5+(-0.5)*Jzz5+m6*rc6z^2+(0.5)*Jxx6+(0.5)*Jyy6+(-0.5)*Jzz6
        Row[56]:
          Index = 55
          Value = 0
          Unit = 
          Description = 
        Row[57]:
          Index = 56
          Value = 0
          Unit = 
          Description = 
        Row[58]:
          Index = 57
          Value = 0
          Unit = 
          Description = 
        Row[59]:
          Index = 58
          Value = 0
          Unit = 
          Description = 
        Row[60]:
          Index = 59
          Value = 0.00052765
          Unit = kgm
          Description = m6*rc6x
        Row[61]:
          Index = 60
          Value = -0.0030867
          Unit = kgm
          Description = m6*rc6y
        Row[62]:
          Index = 61
          Value = 0
          Unit = 
          Description = 
        Row[63]:
          Index = 62
          Value = 5.0962e-05
          Unit = kgm^2
          Description = m6*rc6x*rc6y
        Row[64]:
          Index = 63
          Value = -0.0015762
          Unit = kgm^2
          Description = m6*rc6y*rc6z
        Row[65]:
          Index = 64
          Value = 0.0005846
          Unit = kgm^2
          Description = m6*rc6x*rc6z
        Row[66]:
          Index = 65
          Value = 0.00067399
          Unit = kgm^2
          Description = m6*rc6x^2+(-0.5)*Jxx6+(0.5)*Jyy6+(0.5)*Jzz6
        Row[67]:
          Index = 66
          Value = 0.0013929
          Unit = kgm^2
          Description = m6*rc6y^2+(0.5)*Jxx6+(-0.5)*Jyy6+(0.5)*Jzz6
        Row[68]:
          Index = 67
          Value = 0
          Unit = 
          Description = 
        Row[69]:
          Index = 68
          Value = 0
          Unit = 
          Description = 
        Row[70]:
          Index = 69
          Value = 0
          Unit = 
          Description = 
        Row[71]:
          Index = 70
          Value = 0
          Unit = 
          Description = 
        Row[72]:
          Index = 71
          Value = 0
          Unit = 
          Description = mTool
        Row[73]:
          Index = 72
          Value = 0
          Unit = 
          Description = mTool*rcToolx
        Row[74]:
          Index = 73
          Value = 0
          Unit = 
          Description = mTool*rcTooly
        Row[75]:
          Index = 74
          Value = 0
          Unit = 
          Description = mTool*rcToolz
        Row[76]:
          Index = 75
          Value = 0
          Unit = 
          Description = mTool*rcToolx*rcTooly
        Row[77]:
          Index = 76
          Value = 0
          Unit = 
          Description = mTool*rcTooly*rcToolz
        Row[78]:
          Index = 77
          Value = 0
          Unit = 
          Description = mTool*rcToolx*rcToolz
        Row[79]:
          Index = 78
          Value = 0
          Unit = 
          Description = mTool*rcToolx^2
        Row[80]:
          Index = 79
          Value = 0
          Unit = 
          Description = mTool*rcTooly^2
        Row[81]:
          Index = 80
          Value = 0
          Unit = 
          Description = mTool*rcToolz^2
        Row[82]:
          Index = 81
          Value = 0
          Unit = 
          Description = JxxTool
        Row[83]:
          Index = 82
          Value = 0
          Unit = 
          Description = JyyTool
        Row[84]:
          Index = 83
          Value = 0
          Unit = 
          Description = JzzTool
        Row[85]:
          Index = 84
          Value = 0
          Unit = 
          Description = 
        Row[86]:
          Index = 85
          Value = 0
          Unit = 
          Description = 
        Row[87]:
          Index = 86
          Value = 9.8824e-05
          Unit = kgm^2
          Description = JDrive3
        Row[88]:
          Index = 87
          Value = 5.2689e-05
          Unit = kgm^2
          Description = JDrive4
        Row[89]:
          Index = 88
          Value = 5.129e-05
          Unit = kgm^2
          Description = JDrive5
        Row[90]:
          Index = 89
          Value = 5.2318e-05
          Unit = kgm^2
          Description = JDrive6
        Row[91]:
          Index = 90
          Value = 4.1946
          Unit = Nms
          Description = dV1
        Row[92]:
          Index = 91
          Value = 7.0888
          Unit = Nms
          Description = dV2
        Row[93]:
          Index = 92
          Value = 3.1195
          Unit = Nms
          Description = dV3
        Row[94]:
          Index = 93
          Value = 1.481
          Unit = Nms
          Description = dV4
        Row[95]:
          Index = 94
          Value = 1.1989
          Unit = Nms
          Description = dV5
        Row[96]:
          Index = 95
          Value = 0.67577
          Unit = Nms
          Description = dV6
        Row[97]:
          Index = 96
          Value = 25.5954
          Unit = Nm
          Description = dC1
        Row[98]:
          Index = 97
          Value = 14.3239
          Unit = Nm
          Description = dC2
        Row[99]:
          Index = 98
          Value = 7.6123
          Unit = Nm
          Description = dC3
        Row[100]:
          Index = 99
          Value = 7.9035
          Unit = Nm
          Description = dC4
        Row[101]:
          Index = 100
          Value = 3.5858
          Unit = Nm
          Description = dC5
        Row[102]:
          Index = 101
          Value = 5.2501
          Unit = Nm
          Description = dC6
      CouplingsIsInvisible = 0
      Couplings:
        LinearCoupling[1]:
          SourceAxisIsReadOnly = 1
          SourceAxis = 5
          SourceAxisUnitsIsReadOnly = 1
          SourceAxisUnits = 1.0
          TargetJointAxisIsReadOnly = 1
          TargetJointAxis = 6
          TargetJointAxisUnitsIsReadOnly = 1
          TargetJointAxisUnits = 0.02
      JointAxesPositionLimits:
        JointAxisIsReadOnly = 0
        JointAxis[1] = ConfigureJointAxesLimits
          LowerLimitMin = -170.0
          UpperLimitMax = 170.0
          LowerLimit = -170.0
          UpperLimit = 170.0
        JointAxis[2] = ConfigureJointAxesLimits
          LowerLimitMin = -95.0
          UpperLimitMax = 135.0
          LowerLimit = -95.0
          UpperLimit = 135.0
        JointAxis[3] = ConfigureJointAxesLimits
          LowerLimitMin = -155.0
          UpperLimitMax = 90.0
          LowerLimit = -155.0
          UpperLimit = 90.0
        JointAxis[4] = ConfigureJointAxesLimits
          LowerLimitMin = -200.0
          UpperLimitMax = 200.0
          LowerLimit = -200.0
          UpperLimit = 200.0
        JointAxis[5] = ConfigureJointAxesLimits
          LowerLimitMin = -125.0
          UpperLimitMax = 125.0
          LowerLimit = -125.0
          UpperLimit = 125.0
        JointAxis[6] = ConfigureJointAxesLimits
          LowerLimitMin = -2700.0
          UpperLimitMax = 2700.0
          LowerLimit = -2700.0
          UpperLimit = 2700.0
```

### Config.mppackmlcore - 5APC3100_KBU1_000/mappServices/Config.mppackmlcore
```
Element gPackMLCore (Type=mppackmlcore)
  Core:
    StartupActiveMode = 1
    StartupActiveState = 2
    Auditing = MpAudit
  Modes:
    Mode[1]:
      ModeID = 1
      Name = Auto
      State[5] = 0
      State[13] = 0
      State[14] = 0
    Mode[2]:
      ModeID = 2
      Name = SemiAuto
    Mode[3]:
      ModeID = 3
  Alarms = MpAlarmX
```

### Config_10.mpfilemanagerui - 5APC3100_KBU1_000/mappServices/Config_10.mpfilemanagerui
```
Element gFileManagerUI (Type=mpfilemanagerui)
  Alarms = MpAlarmX
Element gFileManagerUI_R (Type=mpfilemanagerui)
```

### Config_11.mpwebxs - 5APC3100_KBU1_000/mappServices/Config_11.mpwebxs
```
Element WebXs (Type=mpwebxs)
```

### Config_12.mprecipexml - 5APC3100_KBU1_000/mappServices/Config_12.mprecipexml
```
Element gRecipeXml (Type=mprecipexml)
  mapp.Recipe.Xml:
    Auditing = MpAudit
  Alarms = MpAlarmX
```

### Config_14.mpaudittrail - 5APC3100_KBU1_000/mappServices/Config_14.mpaudittrail
```
Element gAuditTrail (Type=mpaudittrail)
  Audit:
    Events:
      [0] = 16
      [1] = 2
      [2] = 18
      [3] = 19
    TextSource = TXT
      Name = 
      OutputFormat = Audit/Event/Root
      Display = Ne
    Export:
      Encrypt = FALSE
  Alarms = MpAlarmX
```

### Config_15.mppackmlmodule - 5APC3100_KBU1_000/mappServices/Config_15.mppackmlmodule
```
Element gPackMLModule (Type=mppackmlmodule)
  Module:
    Parent:
      Parent
      Activation = 0
```

### Config_8.mpalarmxcore - 5APC3100_KBU1_000/mappServices/Config_8.mpalarmxcore
```
Element gAlarmXCore0 (Type=mpalarmxcore)
  mapp.AlarmX.Core.Configuration:
    [0]:
      Name = Error
      Message = Robot Error
      Code = 1
      Behavior = LevelMonitoring
        Monitoring:
          MonitoredPV = ::Alarms:test_error
          HighLimitEnable = Static
            Limit = 0.7
            LimitText = ERROR MAKS NAPRAW
    [1]:
      Name = TooManyBolts
      Message = {&LimitText}
      Code = 111
      Behavior = LevelMonitoring
        Monitoring:
          MonitoredPV = ::DetectedScrew
          LowLimitEnable = Static
            Limit = 0.5
            LimitText = Nie wykryto śrubki
          HighLimitEnable = Static
            Limit = 1.5
            LimitText = Wykryto za dużo śrubek
    [2]:
      Name = TooManyWrenches
      Message = {&LimitText}
      Code = 112
      Behavior = LevelMonitoring
        Monitoring:
          MonitoredPV = ::DetectedWrench
          LowLimitEnable = Static
            Limit = 0.5
            LimitText = Nie wykryto klucza
          HighLimitEnable = Static
            Limit = 1.5
            LimitText = Wykryto za dużo kluczy
    [3]:
      Name = TooManyBoltWashers
      Message = {&LimitText}
      Code = 114
      Behavior = LevelMonitoring
        Monitoring:
          MonitoredPV = ::DetectedScrewWasher
          LowLimitEnable = Static
            Limit = 0.5
            LimitText = Nie wykryto podkładki
          HighLimitEnable = Static
            Limit = 1.5
            LimitText = Wykryto za dużo podkładek
    [4]:
      Name = TooManySquares
      Message = {&LimitText}
      Code = 119
      Behavior = LevelMonitoring
        Monitoring:
          MonitoredPV = ::DetectedSquares
          LowLimitEnable = Static
            Limit = 6.5
            LimitText = Wykryto za mało podstawek
          HighLimitEnable = Static
            Limit = 7.5
            LimitText = Wykryto za dużo podstawek
    [5]:
      Name = HomeERROR
      Message = Home Positions has not been read from retain memory
      Code = 101
      Behavior = LevelMonitoring
        Monitoring:
          MonitoredPV = ::emptyPos
          HighLimitEnable = Static
            Limit = 107
            LimitText =  Retake Homing procedure
    [6]:
      Name = Robot is not Home
      Message = Robot interrupts vision system 
      Code = 111
      Behavior = LevelMonitoring
        Monitoring:
          MonitoredPV = ::MpRoboArm6Axis_0.X
          HighLimitEnable = Static
            Limit = 400
            LimitText = Robot in ROI
```

### Config_9.mpuserx - 5APC3100_KBU1_000/mappServices/Config_9.mpuserx
```
Element UserMgmtX (Type=mpuserx)
  ServerSettings:
    Server:
      AdditionalUserData:
        [0] = mail
        [1] = telephoneNumber
  Users:
    DefUser#1:
      id = admin
      name = Administrator
    DefUser#2:
      id = Anonymous
    DefUser#3:
      id = operator1
  Groups:
    DefGroup#1:
      id = Administrators
      level = 100
      admin = TRUE
      rights:
        [0] = FullAccess
    DefGroup#2:
      id = Operator
      level = 70
      rights:
        [0] = StartOnly
    DefGroup#3:
      id = Everyone
      rights:
        [0] = ViewOnly
```

### viComp.visioncomponent - 5APC3100_KBU1_000/mappVision/viComp.visioncomponent
```
Element gCamera (Type=visioncomponent)
  VisionApplicationReference = PixelCounter
```

## Configuration Config2

CPU 5APC3100.KBU1-000, AutomationRuntime B4.92, Build 4.1.2, Safety 0.0, Vc V4.72.5

### Task classes (Cpu.sw)
```
Cyclic#1 (cycle 2000 us, tolerance 0 us):
  OpcCtrl <- Services.OpcCtrl.prg
  ComauManua <- Robot.PackML.PackML_Manual.prg
  PackML_Aut <- Robot.PackML.PackML_Auto.prg
  PackML_Log <- Robot.PackML.PackML_Logic.prg
  RobotMove <- (binary)
Cyclic#4:
  Alarms <- Services.Alarms.prg
  Elements_d <- Camera.Elements_detection.prg
  PackML_Sem <- Robot.PackML.PackML_SemiAuto.prg
DataObjects: McAcpSys
NcDataObjects: McDriveLog
Binaries: McAcpDrv, udbdef, McAcpSim, mvLoader, arflatprv, McPathXT, TCData, visionUnit, mCoWebSc, McMechSys, FWRules, arcoal, arsvcreg, viApp, Settings, iomap, Config_3, Settings_1, viComp, Config_4, Role, ashwac, Hierarchy, asfw, Config_5, sysconf, Config_2, arconfig, Config_1, ashwd, User, Config_6, Config, Config_7, Config_9, PixelCount, Config_8, Matching15
Libraries: McBase, ViBase, AsZip, FileIO, AsARCfg, powerlnk, AsEPL, AsIO, sys_lib, astime, runtime, MpRobotics, McAxGroup, MpBase, McPathGen, McAxis, McProgInt, McAcpAx, CoTrace, standard, MpAlarmX, MpUserX, asarprof, asieccon, asarlog, asmem, brsystem, dataobj, arssl, asopcuac, aseth, ashw, arcert, aruser
```

### Hardware
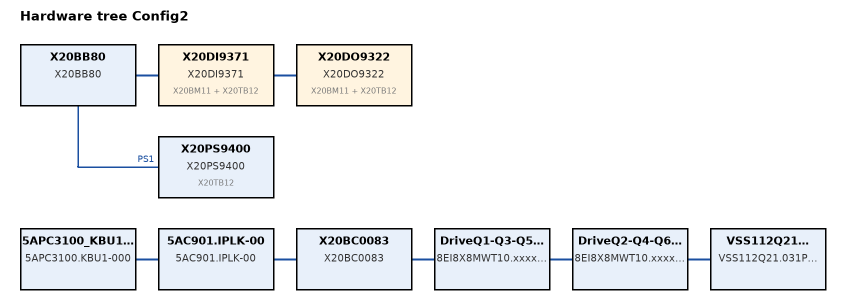
```
5AC901.IPLK-00 : 5AC901.IPLK-00 v1.8.0.1  [SL -> 5APC3100_KBU1_000.SL2]
  Connector IF1:
    MtuSize = 1500
    CycleTime = 400
    Channel1
    ChannelID1 = McAcpBroadcast
    ChannelType1 = OCTET[200]
    InternetAddress = 192.168.200.240
    SubnetMask = 255.255.255.0
5APC3100_KBU1_000 : 5APC3100.KBU1-000 v2.2.1.0
  Connector IF3:
    AssignedOperatingSystem = ARemb
    ActivateDevice = 1
    Mode = Manual
    InternetAddress = 192.168.0.10
    SubnetMask = 255.255.255.0
    ActivateSnmp = 2
  Connector IF4:
    AssignedOperatingSystem = ARemb
    ActivateDevice = 1
  Connector IF5:
    AssignedOperatingSystem = ARemb
  Connector IF6:
    AssignedOperatingSystem = ARemb
  Connector IF7:
    AssignedOperatingSystem = ARemb
  Connector IF8:
    AssignedOperatingSystem = ARemb
  ConfigurationID = RobotComau_Config1
  Simulation = 1
  RemMemDevice = PCI.2.IPLK.SRAM
  RemMemSize = 1024
  PermanentPvSize = 512
  RemanentGlobalPvSize = 512
  TimerDeviceType = EPLX2X
  TimerDevice = 5AC901.IPLK-00.IF1
  TaskClassIdleTime = 2000
  Cyclic1Duration = 2000
  Cyclic1Tolerance = 0
  FileDevice1
  FileDeviceName1 = CNC_PrgDir
  FileDevicePath1 = C:\Users\Szkolenie\Documents\GitHub\Robot-Comau\Logical
  FtpUser1
  FtpUsername1 = admin
  FtpUserPassword1 = QCzPEyxrRcQJkbJUmFYJydudCaTwVAMxyUFRcNQN44M=
  FtpUserSalt1 = 07CFXo9y
  FTPAccessRight1 = 0
  ActivateOpcUa = 1
  OpcUaInformationModels_PV_Version = 1
DriveQ1-Q3-Q5_Racer3_1 : 8EI8X8MWT10.xxxx-1 v2.3.1.1  [PLK1 -> X20BC0083.PLK2 (NodeNumber=4) [Cable Type=PowerlinkCable, Length=10, Version=1.0.0.3]; PLK2 -> DriveQ2-Q4-Q6_Racer3_1.PLK1 (NodeNumber=4) [Cable Type=PowerlinkCable, Length=10, Version=1.0.0.3]]
  DriveConfiguration/Module:
    McAcoposTypeID = AcoposP3TConfig
    ActivateACOPOSSimulationOnPLC = 0
  DriveConfiguration/Encoder/EncoderX41:
    InterfaceType = EnDat
  DriveConfiguration/Encoder/EncoderX42:
    InterfaceType = EnDat
  DriveConfiguration/Encoder/EncoderX43:
    InterfaceType = EnDat
  DriveConfiguration/Channel[1]/RealAxis:
    AxisReference = gAxisQ1_Racer3_1
    MechanicalElementsIsInvisible = 0
  DriveConfiguration/Channel[1]/RealAxis/MechanicalElements/Gearbox:
    InputIsReadOnly = 1
    Input = 81818
    OutputIsReadOnly = 1
    Output = 1000
  DriveConfiguration/Channel[1]/RealAxis/MechanicalElements/RotaryToLinearTransformation:
    ReferenceDistanceIsReadOnly = 1
    ReferenceDistance = 360
  DriveConfiguration/Channel[1]/RealAxis/Controller:
    ModeIsReadOnly = 1
    Mode = PositionControllerWithTorqueFeedForward
  DriveConfiguration/Channel[1]/RealAxis/Controller/Mode/Position:
    ProportionalGainIsReadOnly = 1
    ProportionalGain = 75.0
    IntegrationTimeIsReadOnly = 1
    IntegrationTime = 0.0
    TotalDelayTime = 0.0004
  DriveConfiguration/Channel[1]/RealAxis/Controller/Mode/Speed:
    ProportionalGainIsReadOnly = 1
    ProportionalGain = 2.0
    IntegrationTimeIsReadOnly = 1
    IntegrationTime = 0.0
    FilterTimeIsReadOnly = 1
    FilterTime = 0.0008
  DriveConfiguration/Channel[1]/RealAxis/Controller/Mode:
    FeedForwardIsReadOnly = 1
    FeedForward = CyclicValueFromAxesGroup
  DriveConfiguration/Channel[1]/RealAxis/Controller/Mode/LoopFilters:
    LoopFilterXIsReadOnly = 0
    LoopFilter1 = NotUsed
    LoopFilter2 = NotUsed
    LoopFilter3 = NotUsed
  DriveConfiguration/Channel[1]/RealAxis/Homing:
    ModeIsReadOnly = 0
    Mode = Direct
  DriveConfiguration/Channel[1]/RealAxis/Homing/Mode:
    Position = 0.0
    ReferencePulse = NotUsed
  DriveConfiguration/Channel[1]/RealAxis/Homing:
    RestorePositionVariable = ::RestorePos[0]
  DriveConfiguration/Channel[1]/RealAxis/StopReaction:
    QuickstopIsReadOnly = 0
    Quickstop = DecelerationLimit
    DriveErrorIsReadOnly = 0
    DriveError = DecelerationLimit
  DriveConfiguration/Channel[1]/RealAxis/MovementErrorLimits:
    PositionError = 1.0
    VelocityErrorMonitoring = Automatic1
  DriveConfiguration/Channel[1]/RealAxis:
    JerkFilterIsReadOnly = 0
    JerkFilter = Used
  DriveConfiguration/Channel[1]/RealAxis/JerkFilter:
    JerkTimeMin = 0
    JerkTime = 0.01
  DriveConfiguration/Channel[1]/RealAxis/DigitalInputs/HomingSwitch:
    SourceIsReadOnly = 0
    Source = NotUsed
    Level = High
  DriveConfiguration/Channel[1]/RealAxis/DigitalInputs/PositiveLimitSwitch:
    SourceIsReadOnly = 0
    Source = NotUsed
    Level = High
  DriveConfiguration/Channel[1]/RealAxis/DigitalInputs/NegativeLimitSwitch:
    SourceIsReadOnly = 0
    Source = NotUsed
    Level = High
  DriveConfiguration/Channel[1]/RealAxis/DigitalInputs/Trigger1:
    Source = X8Trigger1
    Level = High
  DriveConfiguration/Channel[1]/RealAxis/DigitalInputs/Trigger2:
    Source = X8Trigger2
    Level = High
  DriveConfiguration/Channel[1]/RealAxis/DigitalInputs/Quickstop:
    Input = Trigger2
  DriveConfiguration/Channel[1]/RealAxis/Simulation:
    SimulationModeOnPLC = SetValueGeneration
    SimulationModeOnACOPOS = NotUsed
  DriveConfiguration/Channel[1]/RealAxis/AxisFeatures:
    FeatureRef[1] = Feature_Brake_Racer3_1
  DriveConfiguration/Channel[1]:
    ExternalEncoderAxis = NotUsed
  DriveConfiguration/Channel[2]/RealAxis:
    AxisReference = gAxisQ3_Racer3_1
    MechanicalElementsIsInvisible = 0
  DriveConfiguration/Channel[2]/RealAxis/MechanicalElements/Gearbox:
    InputIsReadOnly = 1
    Input = 72
    OutputIsReadOnly = 1
    Output = 1
  DriveConfiguration/Channel[2]/RealAxis/MechanicalElements/RotaryToLinearTransformation:
    ReferenceDistanceIsReadOnly = 1
    ReferenceDistance = 360
  DriveConfiguration/Channel[2]/RealAxis/Controller:
    ModeIsReadOnly = 1
    Mode = PositionControllerWithTorqueFeedForward
  DriveConfiguration/Channel[2]/RealAxis/Controller/Mode/Position:
    ProportionalGainIsReadOnly = 1
    ProportionalGain = 50.0
    IntegrationTimeIsReadOnly = 1
    IntegrationTime = 0.0
    TotalDelayTime = 0.0004
  DriveConfiguration/Channel[2]/RealAxis/Controller/Mode/Speed:
    ProportionalGainIsReadOnly = 1
    ProportionalGain = 1.5
    IntegrationTimeIsReadOnly = 1
    IntegrationTime = 0.0
    FilterTimeIsReadOnly = 1
    FilterTime = 0.0008
  DriveConfiguration/Channel[2]/RealAxis/Controller/Mode:
    FeedForwardIsReadOnly = 1
    FeedForward = CyclicValueFromAxesGroup
  DriveConfiguration/Channel[2]/RealAxis/Controller/Mode/LoopFilters:
    LoopFilterXIsReadOnly = 0
    LoopFilter1 = NotUsed
    LoopFilter2 = NotUsed
    LoopFilter3 = NotUsed
  DriveConfiguration/Channel[2]/RealAxis/Homing:
    ModeIsReadOnly = 0
    Mode = Direct
  DriveConfiguration/Channel[2]/RealAxis/Homing/Mode:
    Position = -90
    ReferencePulse = NotUsed
  DriveConfiguration/Channel[2]/RealAxis/Homing:
    RestorePositionVariable = ::RestorePos[2]
  DriveConfiguration/Channel[2]/RealAxis/StopReaction:
    QuickstopIsReadOnly = 0
    Quickstop = DecelerationLimit
    DriveErrorIsReadOnly = 0
    DriveError = DecelerationLimit
  DriveConfiguration/Channel[2]/RealAxis/MovementErrorLimits:
    PositionError = 1.0
    VelocityErrorMonitoring = Automatic1
  DriveConfiguration/Channel[2]/RealAxis:
    JerkFilterIsReadOnly = 0
    JerkFilter = Used
  DriveConfiguration/Channel[2]/RealAxis/JerkFilter:
    JerkTimeMin = 0
    JerkTime = 0.01
  DriveConfiguration/Channel[2]/RealAxis/DigitalInputs/HomingSwitch:
    SourceIsReadOnly = 0
    Source = NotUsed
    Level = High
  DriveConfiguration/Channel[2]/RealAxis/DigitalInputs/PositiveLimitSwitch:
    SourceIsReadOnly = 0
    Source = NotUsed
    Level = High
  DriveConfiguration/Channel[2]/RealAxis/DigitalInputs/NegativeLimitSwitch:
    SourceIsReadOnly = 0
    Source = NotUsed
    Level = High
  DriveConfiguration/Channel[2]/RealAxis/DigitalInputs/Trigger1:
    Source = X8Trigger1
    Level = High
  DriveConfiguration/Channel[2]/RealAxis/DigitalInputs/Trigger2:
    Source = X8Trigger2
    Level = High
  DriveConfiguration/Channel[2]/RealAxis/DigitalInputs/Quickstop:
    Input = Trigger2
  DriveConfiguration/Channel[2]/RealAxis/Simulation:
    SimulationModeOnPLC = SetValueGeneration
    SimulationModeOnACOPOS = NotUsed
  DriveConfiguration/Channel[2]/RealAxis/AxisFeatures:
    FeatureRef[1] = Feature_Brake_Racer3_1
  DriveConfiguration/Channel[2]:
    ExternalEncoderAxis = NotUsed
  DriveConfiguration/Channel[3]/RealAxis:
    AxisReference = gAxisQ5_Racer3_1
    MechanicalElementsIsInvisible = 0
  DriveConfiguration/Channel[3]/RealAxis/MechanicalElements/Gearbox:
    InputIsReadOnly = 1
    Input = 612
    OutputIsReadOnly = 1
    Output = 10
  DriveConfiguration/Channel[3]/RealAxis/MechanicalElements/RotaryToLinearTransformation:
    ReferenceDistanceIsReadOnly = 1
    ReferenceDistance = 360
  DriveConfiguration/Channel[3]/RealAxis/Controller:
    ModeIsReadOnly = 1
    Mode = PositionControllerWithTorqueFeedForward
  DriveConfiguration/Channel[3]/RealAxis/Controller/Mode/Position:
    ProportionalGainIsReadOnly = 1
    ProportionalGain = 200.0
    IntegrationTimeIsReadOnly = 1
    IntegrationTime = 0.0
    TotalDelayTime = 0.0004
  DriveConfiguration/Channel[3]/RealAxis/Controller/Mode/Speed:
    ProportionalGainIsReadOnly = 1
    ProportionalGain = 1.5
    IntegrationTimeIsReadOnly = 1
    IntegrationTime = 0.0
    FilterTimeIsReadOnly = 1
    FilterTime = 0.0008
  DriveConfiguration/Channel[3]/RealAxis/Controller/Mode:
    FeedForwardIsReadOnly = 1
    FeedForward = CyclicValueFromAxesGroup
  DriveConfiguration/Channel[3]/RealAxis/Controller/Mode/LoopFilters:
    LoopFilterXIsReadOnly = 0
    LoopFilter1 = NotUsed
    LoopFilter2 = NotUsed
    LoopFilter3 = NotUsed
  DriveConfiguration/Channel[3]/RealAxis/Homing:
    ModeIsReadOnly = 0
    Mode = Direct
  DriveConfiguration/Channel[3]/RealAxis/Homing/Mode:
    Position = 0.0
    ReferencePulse = NotUsed
  DriveConfiguration/Channel[3]/RealAxis/Homing:
    RestorePositionVariable = ::RestorePos[4]
  DriveConfiguration/Channel[3]/RealAxis/StopReaction:
    QuickstopIsReadOnly = 0
    Quickstop = DecelerationLimit
    DriveErrorIsReadOnly = 0
    DriveError = DecelerationLimit
  DriveConfiguration/Channel[3]/RealAxis/MovementErrorLimits:
    PositionError = 1.0
    VelocityErrorMonitoring = Automatic1
  DriveConfiguration/Channel[3]/RealAxis:
    JerkFilterIsReadOnly = 0
    JerkFilter = Used
  DriveConfiguration/Channel[3]/RealAxis/JerkFilter:
    JerkTimeMin = 0
    JerkTime = 0.01
  DriveConfiguration/Channel[3]/RealAxis/DigitalInputs/HomingSwitch:
    SourceIsReadOnly = 0
    Source = NotUsed
    Level = High
  DriveConfiguration/Channel[3]/RealAxis/DigitalInputs/PositiveLimitSwitch:
    SourceIsReadOnly = 0
    Source = NotUsed
    Level = High
  DriveConfiguration/Channel[3]/RealAxis/DigitalInputs/NegativeLimitSwitch:
    SourceIsReadOnly = 0
    Source = NotUsed
    Level = High
  DriveConfiguration/Channel[3]/RealAxis/DigitalInputs/Trigger1:
    Source = X8Trigger1
    Level = High
  DriveConfiguration/Channel[3]/RealAxis/DigitalInputs/Trigger2:
    Source = X8Trigger2
    Level = High
  DriveConfiguration/Channel[3]/RealAxis/DigitalInputs/Quickstop:
    Input = Trigger2
  DriveConfiguration/Channel[3]/RealAxis/Simulation:
    SimulationModeOnPLC = SetValueGeneration
    SimulationModeOnACOPOS = NotUsed
  DriveConfiguration/Channel[3]/RealAxis/AxisFeatures:
    FeatureRef[1] = Feature_Brake_Racer3_1
  DriveConfiguration/Channel[3]:
    ExternalEncoderAxis = NotUsed
DriveQ2-Q4-Q6_Racer3_1 : 8EI8X8MWT10.xxxx-1 v2.3.1.1  [PLK1 -> DriveQ1-Q3-Q5_Racer3_1.PLK2 (NodeNumber=5) [Cable Type=PowerlinkCable, Length=10, Version=1.0.0.3]; PLK2 -> VSS112Q21.031P-000.PLK2 (NodeNumber=5) [Cable Type=PowerlinkCable, Length=10, Version=1.0.0.3]]
  DriveConfiguration/Module:
    McAcoposTypeID = AcoposP3TConfig
    ActivateACOPOSSimulationOnPLC = 0
  DriveConfiguration/Encoder/EncoderX41:
    InterfaceType = EnDat
  DriveConfiguration/Encoder/EncoderX42:
    InterfaceType = EnDat
  DriveConfiguration/Encoder/EncoderX43:
    InterfaceType = EnDat
  DriveConfiguration/Channel[1]/RealAxis:
    AxisReference = gAxisQ2_Racer3_1
    MechanicalElementsIsInvisible = 0
  DriveConfiguration/Channel[1]/RealAxis/MechanicalElements/Gearbox:
    InputIsReadOnly = 1
    Input = 80
    OutputIsReadOnly = 1
    Output = 1
  DriveConfiguration/Channel[1]/RealAxis/MechanicalElements/RotaryToLinearTransformation:
    ReferenceDistanceIsReadOnly = 1
    ReferenceDistance = 360
  DriveConfiguration/Channel[1]/RealAxis/Controller:
    ModeIsReadOnly = 1
    Mode = PositionControllerWithTorqueFeedForward
  DriveConfiguration/Channel[1]/RealAxis/Controller/Mode/Position:
    ProportionalGainIsReadOnly = 1
    ProportionalGain = 50.0
    IntegrationTimeIsReadOnly = 1
    IntegrationTime = 0.0
    TotalDelayTime = 0.0004
  DriveConfiguration/Channel[1]/RealAxis/Controller/Mode/Speed:
    ProportionalGainIsReadOnly = 1
    ProportionalGain = 2.0
    IntegrationTimeIsReadOnly = 1
    IntegrationTime = 0.0
    FilterTimeIsReadOnly = 1
    FilterTime = 0.0008
  DriveConfiguration/Channel[1]/RealAxis/Controller/Mode:
    FeedForwardIsReadOnly = 1
    FeedForward = CyclicValueFromAxesGroup
  DriveConfiguration/Channel[1]/RealAxis/Controller/Mode/LoopFilters:
    LoopFilterXIsReadOnly = 0
    LoopFilter1 = NotUsed
    LoopFilter2 = NotUsed
    LoopFilter3 = NotUsed
  DriveConfiguration/Channel[1]/RealAxis/Homing:
    ModeIsReadOnly = 0
    Mode = Direct
  DriveConfiguration/Channel[1]/RealAxis/Homing/Mode:
    Position = 0.0
    ReferencePulse = NotUsed
  DriveConfiguration/Channel[1]/RealAxis/Homing:
    RestorePositionVariable = ::RestorePos[1]
  DriveConfiguration/Channel[1]/RealAxis/StopReaction:
    QuickstopIsReadOnly = 0
    Quickstop = DecelerationLimit
    DriveErrorIsReadOnly = 0
    DriveError = DecelerationLimit
  DriveConfiguration/Channel[1]/RealAxis/MovementErrorLimits:
    PositionError = 1.0
    VelocityErrorMonitoring = Automatic1
  DriveConfiguration/Channel[1]/RealAxis:
    JerkFilterIsReadOnly = 0
    JerkFilter = Used
  DriveConfiguration/Channel[1]/RealAxis/JerkFilter:
    JerkTimeMin = 0
    JerkTime = 0.01
  DriveConfiguration/Channel[1]/RealAxis/DigitalInputs/HomingSwitch:
    SourceIsReadOnly = 0
    Source = NotUsed
    Level = High
  DriveConfiguration/Channel[1]/RealAxis/DigitalInputs/PositiveLimitSwitch:
    SourceIsReadOnly = 0
    Source = NotUsed
    Level = High
  DriveConfiguration/Channel[1]/RealAxis/DigitalInputs/NegativeLimitSwitch:
    SourceIsReadOnly = 0
    Source = NotUsed
    Level = High
  DriveConfiguration/Channel[1]/RealAxis/DigitalInputs/Trigger1:
    Source = X8Trigger1
    Level = High
  DriveConfiguration/Channel[1]/RealAxis/DigitalInputs/Trigger2:
    Source = X8Trigger2
    Level = High
  DriveConfiguration/Channel[1]/RealAxis/DigitalInputs/Quickstop:
    Input = Trigger2
  DriveConfiguration/Channel[1]/RealAxis/Simulation:
    SimulationModeOnPLC = SetValueGeneration
    SimulationModeOnACOPOS = NotUsed
  DriveConfiguration/Channel[1]/RealAxis/AxisFeatures:
    FeatureRef[1] = Feature_Brake_Racer3_1
  DriveConfiguration/Channel[1]:
    ExternalEncoderAxis = NotUsed
  DriveConfiguration/Channel[2]/RealAxis:
    AxisReference = gAxisQ4_Racer3_1
    MechanicalElementsIsInvisible = 0
  DriveConfiguration/Channel[2]/RealAxis/MechanicalElements/Gearbox:
    InputIsReadOnly = 1
    Input = 612
    OutputIsReadOnly = 1
    Output = 10
  DriveConfiguration/Channel[2]/RealAxis/MechanicalElements/RotaryToLinearTransformation:
    ReferenceDistanceIsReadOnly = 1
    ReferenceDistance = 360
  DriveConfiguration/Channel[2]/RealAxis/Controller:
    ModeIsReadOnly = 1
    Mode = PositionControllerWithTorqueFeedForward
  DriveConfiguration/Channel[2]/RealAxis/Controller/Mode/Position:
    ProportionalGainIsReadOnly = 1
    ProportionalGain = 100.0
    IntegrationTimeIsReadOnly = 1
    IntegrationTime = 0.0
    TotalDelayTime = 0.0004
  DriveConfiguration/Channel[2]/RealAxis/Controller/Mode/Speed:
    ProportionalGainIsReadOnly = 1
    ProportionalGain = 2.0
    IntegrationTimeIsReadOnly = 1
    IntegrationTime = 0.0
    FilterTimeIsReadOnly = 1
    FilterTime = 0.0008
  DriveConfiguration/Channel[2]/RealAxis/Controller/Mode:
    FeedForwardIsReadOnly = 1
    FeedForward = CyclicValueFromAxesGroup
  DriveConfiguration/Channel[2]/RealAxis/Controller/Mode/LoopFilters:
    LoopFilterXIsReadOnly = 0
    LoopFilter1 = NotUsed
    LoopFilter2 = NotUsed
    LoopFilter3 = NotUsed
  DriveConfiguration/Channel[2]/RealAxis/Homing:
    ModeIsReadOnly = 0
    Mode = Direct
  DriveConfiguration/Channel[2]/RealAxis/Homing/Mode:
    Position = 0.0
    ReferencePulse = NotUsed
  DriveConfiguration/Channel[2]/RealAxis/Homing:
    RestorePositionVariable = ::RestorePos[3]
  DriveConfiguration/Channel[2]/RealAxis/StopReaction:
    QuickstopIsReadOnly = 0
    Quickstop = DecelerationLimit
    DriveErrorIsReadOnly = 0
    DriveError = DecelerationLimit
  DriveConfiguration/Channel[2]/RealAxis/MovementErrorLimits:
    PositionError = 1.0
    VelocityErrorMonitoring = Automatic1
  DriveConfiguration/Channel[2]/RealAxis:
    JerkFilterIsReadOnly = 0
    JerkFilter = Used
  DriveConfiguration/Channel[2]/RealAxis/JerkFilter:
    JerkTimeMin = 0
    JerkTime = 0.01
  DriveConfiguration/Channel[2]/RealAxis/DigitalInputs/HomingSwitch:
    SourceIsReadOnly = 0
    Source = NotUsed
    Level = High
  DriveConfiguration/Channel[2]/RealAxis/DigitalInputs/PositiveLimitSwitch:
    SourceIsReadOnly = 0
    Source = NotUsed
    Level = High
  DriveConfiguration/Channel[2]/RealAxis/DigitalInputs/NegativeLimitSwitch:
    SourceIsReadOnly = 0
    Source = NotUsed
    Level = High
  DriveConfiguration/Channel[2]/RealAxis/DigitalInputs/Trigger1:
    Source = X8Trigger1
    Level = High
  DriveConfiguration/Channel[2]/RealAxis/DigitalInputs/Trigger2:
    Source = X8Trigger2
    Level = High
  DriveConfiguration/Channel[2]/RealAxis/DigitalInputs/Quickstop:
    Input = Trigger2
  DriveConfiguration/Channel[2]/RealAxis/Simulation:
    SimulationModeOnPLC = SetValueGeneration
    SimulationModeOnACOPOS = NotUsed
  DriveConfiguration/Channel[2]/RealAxis/AxisFeatures:
    FeatureRef[1] = Feature_Brake_Racer3_1
  DriveConfiguration/Channel[2]:
    ExternalEncoderAxis = NotUsed
  DriveConfiguration/Channel[3]/RealAxis:
    AxisReference = gAxisQ6_Racer3_1
    MechanicalElementsIsInvisible = 0
  DriveConfiguration/Channel[3]/RealAxis/MechanicalElements/Gearbox:
    InputIsReadOnly = 1
    Input = 40
    OutputIsReadOnly = 1
    Output = 1
  DriveConfiguration/Channel[3]/RealAxis/MechanicalElements/RotaryToLinearTransformation:
    ReferenceDistanceIsReadOnly = 1
    ReferenceDistance = 360
  DriveConfiguration/Channel[3]/RealAxis/Controller:
    ModeIsReadOnly = 1
    Mode = PositionControllerWithTorqueFeedForward
  DriveConfiguration/Channel[3]/RealAxis/Controller/Mode/Position:
    ProportionalGainIsReadOnly = 1
    ProportionalGain = 200.0
    IntegrationTimeIsReadOnly = 1
    IntegrationTime = 0.0
    TotalDelayTime = 0.0004
  DriveConfiguration/Channel[3]/RealAxis/Controller/Mode/Speed:
    ProportionalGainIsReadOnly = 1
    ProportionalGain = 1.5
    IntegrationTimeIsReadOnly = 1
    IntegrationTime = 0.0
    FilterTimeIsReadOnly = 1
    FilterTime = 0.0008
  DriveConfiguration/Channel[3]/RealAxis/Controller/Mode:
    FeedForwardIsReadOnly = 1
    FeedForward = CyclicValueFromAxesGroup
  DriveConfiguration/Channel[3]/RealAxis/Controller/Mode/LoopFilters:
    LoopFilterXIsReadOnly = 0
    LoopFilter1 = NotUsed
    LoopFilter2 = NotUsed
    LoopFilter3 = NotUsed
  DriveConfiguration/Channel[3]/RealAxis/Homing:
    ModeIsReadOnly = 0
    Mode = Direct
  DriveConfiguration/Channel[3]/RealAxis/Homing/Mode:
    Position = 0.0
    ReferencePulse = NotUsed
  DriveConfiguration/Channel[3]/RealAxis/Homing:
    RestorePositionVariable = ::RestorePos[5]
  DriveConfiguration/Channel[3]/RealAxis/StopReaction:
    QuickstopIsReadOnly = 0
    Quickstop = DecelerationLimit
    DriveErrorIsReadOnly = 0
    DriveError = DecelerationLimit
  DriveConfiguration/Channel[3]/RealAxis/MovementErrorLimits:
    PositionError = 1.0
    VelocityErrorMonitoring = Automatic1
  DriveConfiguration/Channel[3]/RealAxis:
    JerkFilterIsReadOnly = 0
    JerkFilter = Used
  DriveConfiguration/Channel[3]/RealAxis/JerkFilter:
    JerkTimeMin = 0
    JerkTime = 0.01
  DriveConfiguration/Channel[3]/RealAxis/DigitalInputs/HomingSwitch:
    SourceIsReadOnly = 0
    Source = NotUsed
    Level = High
  DriveConfiguration/Channel[3]/RealAxis/DigitalInputs/PositiveLimitSwitch:
    SourceIsReadOnly = 0
    Source = NotUsed
    Level = High
  DriveConfiguration/Channel[3]/RealAxis/DigitalInputs/NegativeLimitSwitch:
    SourceIsReadOnly = 0
    Source = NotUsed
    Level = High
  DriveConfiguration/Channel[3]/RealAxis/DigitalInputs/Trigger1:
    Source = X8Trigger1
    Level = High
  DriveConfiguration/Channel[3]/RealAxis/DigitalInputs/Trigger2:
    Source = X8Trigger2
    Level = High
  DriveConfiguration/Channel[3]/RealAxis/DigitalInputs/Quickstop:
    Input = Trigger2
  DriveConfiguration/Channel[3]/RealAxis/Simulation:
    SimulationModeOnPLC = SetValueGeneration
    SimulationModeOnACOPOS = NotUsed
  DriveConfiguration/Channel[3]/RealAxis/AxisFeatures:
    FeatureRef[1] = Feature_Brake_Racer3_1
  DriveConfiguration/Channel[3]:
    ExternalEncoderAxis = NotUsed
VSS112Q21.031P-000 : VSS112Q21.031P-000 v1.6.0.543  [PLK2 -> DriveQ2-Q4-Q6_Racer3_1.PLK2 (NodeNumber=6) [Cable Type=PowerlinkCable, Length=10, Version=1.0.0.3]]
  VisionConfig = gCamera
X20BB80 : X20BB80 v1.1.0.0
X20BC0083 : X20BC0083 v2.12.0.0  [PLK1 -> 5AC901.IPLK-00.IF1 (NodeNumber=3) [Cable Type=PowerlinkCable, Length=10, Version=1.0.0.3]; PLK2 -> DriveQ1-Q3-Q5_Racer3_1.PLK1 (NodeNumber=3) [Cable Type=PowerlinkCable, Length=10, Version=1.0.0.3]; SL -> X20BB80.SL1]
X20BM11 : X20BM11 v1.1.0.0  [X2X1 -> X20BB80.IF1]
X20BM11a : X20BM11 v1.1.0.0  [X2X1 -> X20BM11.X2X2]
X20DI9371 : X20DI9371 v1.3.0.0  [SS1 -> X20TB12a.SS; SL -> X20BM11.SL1]
X20DO9322 : X20DO9322 v1.4.0.0  [SS1 -> X20TB12b.SS; SL -> X20BM11a.SL1]
X20PS9400 : X20PS9400 v1.7.0.0  [SS1 -> X20TB12.SS; PS -> X20BB80.PS1]
X20TB12 : X20TB12 v1.0.0.0
X20TB12a : X20TB12 v1.0.0.0
X20TB12b : X20TB12 v1.0.0.0
```

### Cpu.per - 5APC3100_KBU1_000/Cpu.per
```iecst
VAR_CONFIG
	RestorePos AT %M0; (* *)
END_VAR
```

### IoMap.iom - 5APC3100_KBU1_000/IoMap.iom
```iecst
VAR_CONFIG
	::Elements_d:Camera_0.ImageAcq AT %QX."VSS112Q21.031P-000".ImageAcquisition;
	::Elements_d:Camera_0.PixelCntSquareArray[0] AT %ID."VSS112Q21.031P-000".FoundedPixelsNum01;
	::Elements_d:Camera_0.PixelCntSquareArray[1] AT %ID."VSS112Q21.031P-000".FoundedPixelsNum02;
	::Elements_d:Camera_0.PixelCntSquareArray[2] AT %ID."VSS112Q21.031P-000".FoundedPixelsNum03;
	::Elements_d:Camera_0.PixelCntSquareArray[3] AT %ID."VSS112Q21.031P-000".FoundedPixelsNum04;
	::Elements_d:Camera_0.PixelCntSquareArray[4] AT %ID."VSS112Q21.031P-000".FoundedPixelsNum05;
	::Elements_d:Camera_0.PixelCntSquareArray[5] AT %ID."VSS112Q21.031P-000".FoundedPixelsNum06;
	::Elements_d:Camera_0.PixelCntSquareArray[6] AT %ID."VSS112Q21.031P-000".FoundedPixelsNum07;
	::Elements_d:Camera_0.PixelCntSquareArray[7] AT %ID."VSS112Q21.031P-000".FoundedPixelsNum08;
	::Elements_d:Camera_0.PixelCntSquareArray[8] AT %ID."VSS112Q21.031P-000".FoundedPixelsNum09;
	::Elements_d:Camera_0.PixelCntSquareArray[9] AT %ID."VSS112Q21.031P-000".FoundedPixelsNum10;
	::Elements_d:Camera_0.PixelCntSquareArray[10] AT %ID."VSS112Q21.031P-000".FoundedPixelsNum11;
	::Elements_d:Camera_0.PixelCntSquareArray[11] AT %ID."VSS112Q21.031P-000".FoundedPixelsNum12;
	::Elements_d:Camera_0.PixelCntSquareArray[12] AT %ID."VSS112Q21.031P-000".FoundedPixelsNum13;
	::Elements_d:Camera_0.PixelCntSquareArray[13] AT %ID."VSS112Q21.031P-000".FoundedPixelsNum14;
	::Elements_d:Camera_0.Focus AT %QW."VSS112Q21.031P-000".SetFocus;
	::Elements_d:Camera_0.ExposureTime AT %QD."VSS112Q21.031P-000".ExposureTime01;
	::Elements_d:Camera_0.Enable AT %QX."VSS112Q21.031P-000".EnableVF1;
	::Elements_d:Camera_0.NumSearch AT %QB."VSS112Q21.031P-000".NumSearch;
	::Elements_d:Camera_0.Ready AT %IX."VSS112Q21.031P-000".ImageAcquisitionReady;
	::Elements_d:Camera_0.FlashColor AT %QB."VSS112Q21.031P-000".FlashColor01;
	::Elements_d:Camera_0.FlashSegment AT %QB."VSS112Q21.031P-000".FlashSegment01;
	::Elements_d:Camera_0.ModelNumArray[0] AT %IB."VSS112Q21.031P-000".ModelNum01;
	::Elements_d:Camera_0.ModelNumArray[1] AT %IB."VSS112Q21.031P-000".ModelNum02;
	::Elements_d:Camera_0.ModelNumArray[2] AT %IB."VSS112Q21.031P-000".ModelNum03;
	::Elements_d:Camera_0.ModelNumArray[3] AT %IB."VSS112Q21.031P-000".ModelNum04;
	::Elements_d:Camera_0.ModelNumArray[4] AT %IB."VSS112Q21.031P-000".ModelNum05;
	::Elements_d:Camera_0.ModelNumArray[5] AT %IB."VSS112Q21.031P-000".ModelNum06;
	::Elements_d:Camera_0.ModelNumArray[6] AT %IB."VSS112Q21.031P-000".ModelNum07;
	::Elements_d:Camera_0.ModelNumArray[7] AT %IB."VSS112Q21.031P-000".ModelNum08;
	::Elements_d:Camera_0.ModelNumArray[8] AT %IB."VSS112Q21.031P-000".ModelNum09;
	::Elements_d:Camera_0.ModelNumArray[9] AT %IB."VSS112Q21.031P-000".ModelNum10;
	::Elements_d:Camera_0.ModelNumArray[10] AT %IB."VSS112Q21.031P-000".ModelNum11;
	::Elements_d:Camera_0.ModelNumArray[11] AT %IB."VSS112Q21.031P-000".ModelNum12;
	::Elements_d:Camera_0.ModelNumArray[12] AT %IB."VSS112Q21.031P-000".ModelNum13;
	::Elements_d:Camera_0.ModelNumArray[13] AT %IB."VSS112Q21.031P-000".ModelNum14;
	::Comau:doMagnet AT %QX."X20DO9322".DigitalOutput05;
END_VAR
```

### Config_4.axesgroupfeature - 5APC3100_KBU1_000/mappMotion/Comau_Racer3_1/Config_4.axesgroupfeature
```
Element Feature_Programs_Racer3_1 (Type=axesgroupfeature)
  Type = Program
    ModalDataBehaviour = UseAxesGroupSettings
    InitialSettings:
      InterpolationTypes = LinearRapid
      PositionCoordinates = Absolute
      CircleCoordinates = Relative
      JACS_ACSProgramming = JACS
      ContourConnection = Inactive
      ProgrammingUnits = UseAxesGroupSettings
      Feedrates:
        FeedPath = Standard
        FeedCharacteristic = StandardCharacteristic
        FeedType = Feedrate
        FeedReduction = Inactive
        FeedrateValue = 0.0
        InverseFeedrateValue = 0.0
        FeedratePerRevValue = 0.0
    DefaultLanguage = BRGCode
    Location = Default
      FileDevice = CNC_PrgDir
Element Feature_FeedForward_Racer3_1 (Type=axesgroupfeature)
  Type = FeedForward
    Mode = ComputeAndTransmit
    RiseTime = 0.25
    Filter = NotUsed
Element Feature_Jogging_Racer3_1 (Type=axesgroupfeature)
  Type = Jogging
Element Feature_SharedBrakesSignals_Racer3_1 (Type=axesgroupfeature)
  Type = SharedBrakesSignals
    BrakeComposite[1]:
      Axes:
        AxisRef[1] = gAxisQ1_Racer3_1
        AxisRef[2] = gAxisQ2_Racer3_1
        AxisRef[3] = gAxisQ3_Racer3_1
      ErrorBehavior = CloseAfterStop
      Output = Axis
        AxisRef = gAxisQ1_Racer3_1
      Feedback = TimeBased
    BrakeComposite[2]:
      Axes:
        AxisRef[1] = gAxisQ4_Racer3_1
        AxisRef[2] = gAxisQ5_Racer3_1
        AxisRef[3] = gAxisQ6_Racer3_1
      ErrorBehavior = CloseAfterStop
      Output = Axis
        AxisRef = gAxisQ4_Racer3_1
      Feedback = TimeBased
```

### Config_7.axesgroupfeature - 5APC3100_KBU1_000/mappMotion/Config_7.axesgroupfeature
```
Element Feature_WorkspaceMonitoring (Type=axesgroupfeature)
  Type = WorkspaceMonitoring
    ModalDataBehaviour = UseAxesGroupSettings
    WorkspaceRef = Workspace_1
    SelfCollisionDetection = Enabled
    FlangeWorkspace = NotUsed
```

### Config.mppackmlcore - 5APC3100_KBU1_000/mappServices/Config.mppackmlcore
```
Element gPackMLCore (Type=mppackmlcore)
  Core:
    StartupActiveMode = 1
    StartupActiveState = 2
  Modes:
    Mode[1]:
      ModeID = 1
      Name = Auto
      State[1] = 0
      State[5] = 0
      State[8] = 0
      State[9] = 0
      State[10] = 0
      State[11] = 0
      State[12] = 0
      State[13] = 0
      State[14] = 0
    Mode[2]:
      ModeID = 2
      Name = Semiauto
    Mode[3]:
      ModeID = 3
```

### Config_8.mpalarmxcore - 5APC3100_KBU1_000/mappServices/Config_8.mpalarmxcore
```
Element gAlarmXCore0 (Type=mpalarmxcore)
  mapp.AlarmX.Core.Configuration:
    [0]:
      Name = Error
      Message = ERROR
      Code = 1
      Behavior = LevelMonitoring
        Monitoring:
          MonitoredPV = ::Comau:MpRoboArm6Axis_0.Error
          HighLimitEnable = Static
            Limit = 0.7
            LimitText = ERROR MAKS NAPRAW
```

## Logical view

Binary libraries used (declarations not repeated): operator, runtime, astime, AsIecCon, McBase, ViBase 5.18.0, AsZip, FileIO, AsARCfg, powerlnk, AsEPL, AsIO, sys_lib, MpRobotics 5.18.1, McAxGroup 5.18.1, MpBase, McPathGen 5.18.1, McAxis, McProgInt 5.18.1, McAcpAx, CoTrace, standard, AsOpcUac, MpAlarmX, MpUserX, MpFile, AsBrStr, AsArSdm, MpRecipe, MpAudit, MpPackML, MpServer, MpWebXs 5.18.0

### Global.typ - Global data types
```iecst
TYPE
	CameraStruct : 	STRUCT
		ExposureTime : UDINT := 30000;
		Focus : UINT := 30000;
		NumSearch : USINT;
		Enable : BOOL;
		diTrigger : BOOL;
		ImageAcq : BOOL;
		PixelCntSquareArray : ARRAY[0..13]OF UDINT;
		Ready : BOOL;
		FlashColor : USINT;
		ModelNumArray : ARRAY[0..13]OF USINT;
		FlashSegment : USINT;
		prevImgProcessingActive : BOOL;
		ImgProcessingActive : BOOL;
	END_STRUCT;
	PixelCounterLimits : 	STRUCT
		WrenchLimit : UDINT;
		WasherBoltLimit : UDINT;
		ScrewLimit : UDINT;
		HolderLimit : UDINT;
	END_STRUCT;
	gSafeType : 	STRUCT
		diEStop : BOOL;
		diEStopPanel : BOOL;
		diGuardDoor1 : BOOL;
		diGuardDoor2 : BOOL;
		EStop : BOOL;
		EStopPanel : BOOL;
		GuardingDoor : BOOL;
		SafeChannelOK1 : BOOL;
		SafeChannelOK2 : BOOL;
		doAcoposEnable1 : BOOL;
		doAcoposEnable2 : BOOL;
		CommunicationError : BOOL;
		ComErrorAck : BOOL;
	END_STRUCT;
END_TYPE
```

### Global.var - Global variables
```iecst
VAR
	A : McAxisTargetType := (JointAxis:=[0,0,-90,0,90,0],SlaveAxis:=[100]); (*Home value with tool faced torwards floor*)
	Aim1 : ARRAY[0..13] OF BOOL; (*defines aim pose of object number 1*)
	Aim2 : ARRAY[0..13] OF BOOL; (*defines aim pose of object number 2*)
	Aim4 : ARRAY[0..13] OF BOOL; (*defines aim pose of object number 4*)
	Camera_0 : CameraStruct; (*camera*)
	DemoY : INT; (*(DEMO)is used to help with selecting poses at DEMO*)
	DetectedScrew : USINT;
	DetectedScrewWasher : USINT;
	DetectedSquares : USINT; (*swuare detaction*)
	Axis  : USINT;
	DetectedWrench : USINT;
	diDemo : BOOL; (*enables demo mode*)
	doMagnet : BOOL; (*MAgnet contorl*)
	doVisError : BOOL; (*vision error output*)
	gActPos : ARRAY[0..13] OF INT := [2(0),1,2(0),2,0,4,6(0)]; (*table of actual positions of elements *)
	gAimPos : ARRAY[0..13] OF INT := [5(0),1,0,2,5(0),4]; (*target  positions *)
	gAimPos1 : {REDUND_UNREPLICABLE} ARRAY[0..13] OF INT := [5(0),1,0,2,5(0),4]; (*copy of target positions that are modyfied during program *)
	gElementsArray : ARRAY[0..13] OF USINT;
	gIsPosGood : ARRAY[0..13] OF BOOL := [11(0),3(1)]; (*vision system feedback that tells if there is a black pad *)
	gPosBuffor : ARRAY[0..13] OF BOOL; (*positions that can be used as buffor *)
END_VAR
VAR CONSTANT
	gWait : REAL := 0.5;
	gRobPos : ARRAY[0..13] OF McPointType := [(Pos:=(X:=515,Y:=280,Z:=68),Orient:=(Angle1:=0,Angle2:=180,Angle3:=0)),(Pos:=(X:=515,Y:=195,Z:=68),Orient:=(Angle1:=0,Angle2:=180)),(Pos:=(X:=515,Y:=95,Z:=68),Orient:=(Angle1:=0,Angle2:=180,Angle3:=0)),(Pos:=(X:=515,Y:=-5,Z:=68),Orient:=(Angle1:=0,Angle2:=180,Angle3:=0)),(Pos:=(X:=515,Y:=-105,Z:=68),Orient:=(Angle1:=0,Angle2:=180,Angle3:=0)),(Pos:=(X:=515,Y:=-205,Z:=68),Orient:=(Angle1:=0,Angle2:=180)),(Pos:=(X:=515,Y:=-280,Z:=68),Orient:=(Angle1:=0,Angle2:=180,Angle3:=0)),(Pos:=(X:=410,Y:=295,Z:=68),Orient:=(Angle1:=0,Angle2:=180)),(Pos:=(X:=410,Y:=195,Z:=68),Orient:=(Angle1:=0,Angle2:=180)),(Pos:=(X:=410,Y:=95,Z:=68),Orient:=(Angle1:=0,Angle2:=180,Angle3:=0)),(Pos:=(X:=410,Y:=-5,Z:=68),Orient:=(Angle1:=0,Angle2:=180,Angle3:=0)),(Pos:=(X:=410,Y:=-105,Z:=68),Orient:=(Angle1:=0,Angle2:=180,Angle3:=0)),(Pos:=(X:=410,Y:=-205,Z:=68),Orient:=(Angle1:=0,Angle2:=180,Angle3:=0)),(Pos:=(X:=410,Y:=-300,Z:=68),Orient:=(Angle1:=0,Angle2:=180,Angle3:=0))]; (*predefined robot positions*)
END_VAR
VAR
	gSafety : gSafeType; (*safety*)
	gSquareArray : ARRAY[0..13] OF BOOL; (*1 IF is square in i position*)
	gSwapFlag : BOOL; (*enables swap mode *)
	gSwapMap : ARRAY[0..13] OF BOOL; (*(SWAP) Pleaces that can be used to swap*)
	gSwapPoses : ARRAY[0..2] OF McPointType; (*(SWAP) table of positions that will be used to swap procedure*)
END_VAR
VAR CONSTANT
	HOME : McPointType := (Pos:=(X:=435.9,Y:=0,Z:=685),Orient:=(Angle1:=0,Angle2:=90,Angle3:=0)); (*Home pose *)
END_VAR
VAR
	i : USINT;
	Index : ARRAY[0..2] OF INT := [1,2,4]; (*defines order of moves *)
END_VAR
VAR CONSTANT
	LowSpeed : UDINT := 10000;
END_VAR
VAR
	gCompliteFlag : BOOL;
END_VAR
VAR CONSTANT
	MaxSpeed : UDINT := 20000;
END_VAR
VAR
	MpPackMLCore_0 : MpPackMLCore; (*PACK ML*)
	MpPackMLMode_Auto : MpPackMLMode; (*PACK ML AUTO*)
	MpPackMLMode_Manual : MpPackMLMode; (*PACK ML MANUAL*)
	MpPackMLMode_SemiAuto : MpPackMLMode; (*PACK ML SEMIAUTO*)
	P0 : McPointType := (Pos:=(X:=435,Y:=0,Z:=405),Orient:=(Angle1:=0,Angle2:=180,Angle3:=0));
	P1 : McPointType := (Pos:=(X:=510,Y:=-280,Z:=70),Orient:=(Angle1:=0,Angle2:=180,Angle3:=0)); (*first robot position *)
	P1up : McPointType := (Pos:=(X:=510,Y:=-280,Z:=120),Orient:=(Angle1:=0,Angle2:=180,Angle3:=0)); (*position over first robot position*)
	P2 : McPointType := (Pos:=(X:=410,Y:=200,Z:=70),Orient:=(Angle1:=0,Angle2:=180,Angle3:=0)); (*second robot position*)
	P2up : McPointType := (Pos:=(X:=410,Y:=200,Z:=120),Orient:=(Angle1:=0,Angle2:=180,Angle3:=0)); (*position over second robot  position*)
	PixelRange_0 : PixelCounterLimits;
	pom : ARRAY[0..13] OF BOOL;
	PZ : McPointType := (Pos:=(X:=435,Y:=0,Z:=685),Orient:=(Angle1:=0,Angle2:=90,Angle3:=0));
END_VAR
VAR RETAIN
	RestorePos : ARRAY[0..5] OF McAcpAxRestorePosType; (*Comau Home Position*)
END_VAR
VAR
	y : USINT; (*is used to execute moves *)
	emptyPos : USINT;
	gSwapEnable : ARRAY[0..13] OF BOOL; (*list of targets that can be swaped*)
	z : INT;
	gDemoActPos : ARRAY[0..13] OF INT;
END_VAR
```

### Package Logical/Libraries - Global libraries

- Visualisation Logical/mappView (not shown)

### Program Logical/Robot/Recipe (IEC)

#### Variables.var
```iecst
VAR
	WrenchPosible : BOOL;
	Wrench : BOOL;
	testString : STRING[200] := '{"specRows": [ {"from":0, "to":3, "visible":true}, {"from":4, "to":49, "visible":false}]}';
	tempString : STRING[200];
	tableShowLimit : INT;
	tableConfig : STRING[200];
	tabInfo : TabInfo;
	ScrewWasherPosible : BOOL;
	ScrewWasher : BOOL;
	ScrewPosible : BOOL;
	Screw : BOOL;
	PriorytetW : INT;
	PriorytetSW : INT;
	PriorytetS : INT;
	name2 : STRING[80];
	name : STRING[80];
	MpRecipeXml_0 : MpRecipeXml;
	MpRecipeRegPar_0 : MpRecipeRegPar;
	MpFileMngSetup : MpFileManagerUISetupType;
	MpFileMngConnectR : MpFileManagerUIConnectType;
	MpFileManagerUI_R : MpFileManagerUI;
	messageType : STRING[80];
	makeWarning : USINT;
	iFile : INT;
	i : INT;
	clear : BOOL;
END_VAR
```
